Yaskawa INFORM job: A_ROOF_SIDE_0617_2_PAINT_60.JBI

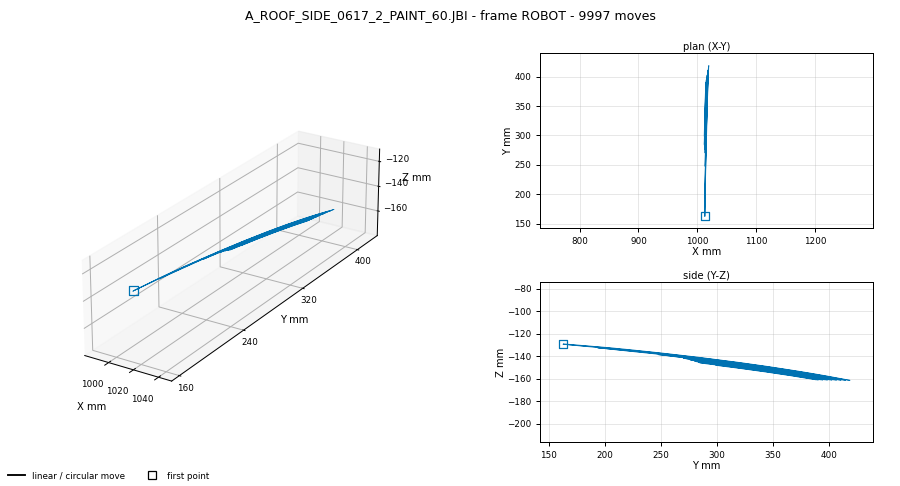
[picture p0: tool path of A_ROOF_SIDE_0617_2_PAINT_60.JBI in frame ROBOT, 9997 of 9997 moves have a stored position in this frame; points joined in program order, loops and branches not executed]
/JOB
//NAME A_ROOF_SIDE_0617_2_PAINT60
//POS
///NPOS 9997,0,0,0,0,0
///TOOL 1
///USER 0
///POSTYPE ROBOT
///RECTAN
///RCONF 1,0,0,0,0,0,0,0,0,0,0,0,0,0,0,0,0,0,0,0,0,0,0,0
C00000=1012.766,163.201,-128.936,166.543,56.945,160.429
C00001=1012.769,163.450,-128.956,166.546,56.934,160.427
C00002=1012.773,163.699,-128.974,166.549,56.922,160.426
C00003=1012.776,163.949,-128.994,166.553,56.910,160.424
C00004=1012.781,164.198,-129.014,166.556,56.898,160.423
C00005=1012.783,164.447,-129.033,166.560,56.886,160.421
C00006=1012.788,164.696,-129.052,166.563,56.875,160.420
C00007=1012.791,164.945,-129.072,166.568,56.863,160.418
C00008=1012.795,165.195,-129.092,166.571,56.851,160.417
C00009=1012.798,165.444,-129.111,166.574,56.839,160.415
C00010=1012.802,165.693,-129.131,166.578,56.827,160.414
C00011=1012.806,165.942,-129.150,166.581,56.815,160.412
C00012=1012.810,166.191,-129.170,166.586,56.803,160.411
C00013=1012.813,166.441,-129.189,166.589,56.791,160.409
C00014=1012.817,166.690,-129.209,166.592,56.779,160.408
C00015=1012.820,166.939,-129.229,166.596,56.767,160.406
C00016=1012.825,167.188,-129.248,166.599,56.756,160.405
C00017=1012.828,167.437,-129.267,166.604,56.743,160.403
C00018=1012.832,167.686,-129.287,166.607,56.732,160.402
C00019=1012.836,167.936,-129.307,166.610,56.720,160.400
C00020=1012.839,168.185,-129.327,166.614,56.707,160.398
C00021=1012.843,168.434,-129.346,166.617,56.695,160.397
C00022=1012.846,168.684,-129.365,166.621,56.683,160.395
C00023=1012.851,168.933,-129.385,166.624,56.671,160.394
C00024=1012.854,169.182,-129.405,166.629,56.659,160.393
C00025=1012.858,169.431,-129.425,166.632,56.647,160.391
C00026=1012.862,169.680,-129.444,166.636,56.635,160.390
C00027=1012.866,169.930,-129.464,166.639,56.623,160.388
C00028=1012.870,170.208,-129.486,166.644,56.609,160.386
C00029=1012.874,170.487,-129.508,166.648,56.596,160.385
C00030=1012.878,170.766,-129.530,166.652,56.583,160.383
C00031=1012.882,171.045,-129.552,166.656,56.569,160.381
C00032=1012.887,171.294,-129.572,166.661,56.557,160.380
C00033=1012.890,171.543,-129.592,166.664,56.545,160.378
C00034=1012.894,171.793,-129.611,166.668,56.532,160.377
C00035=1012.898,172.042,-129.631,166.671,56.521,160.375
C00036=1012.902,172.292,-129.651,166.675,56.509,160.374
C00037=1012.906,172.541,-129.670,166.678,56.497,160.372
C00038=1012.910,172.790,-129.690,166.683,56.485,160.371
C00039=1012.913,173.040,-129.710,166.687,56.472,160.369
C00040=1012.917,173.288,-129.729,166.690,56.460,160.367
C00041=1012.921,173.537,-129.749,166.694,56.448,160.366
C00042=1012.925,173.786,-129.769,166.699,56.436,160.365
C00043=1012.928,174.036,-129.789,166.701,56.424,160.363
C00044=1012.932,174.285,-129.809,166.706,56.411,160.361
C00045=1012.936,174.534,-129.828,166.710,56.399,160.360
C00046=1012.940,174.783,-129.849,166.713,56.388,160.358
C00047=1012.944,175.032,-129.868,166.717,56.375,160.357
C00048=1012.948,175.282,-129.888,166.721,56.363,160.355
C00049=1012.952,175.531,-129.908,166.725,56.351,160.354
C00050=1012.956,175.780,-129.928,166.729,56.339,160.352
C00051=1012.960,176.030,-129.948,166.733,56.326,160.351
C00052=1012.964,176.279,-129.967,166.737,56.314,160.349
C00053=1012.968,176.527,-129.988,166.741,56.302,160.348
C00054=1012.972,176.776,-130.007,166.744,56.289,160.346
C00055=1012.976,177.026,-130.027,166.749,56.277,160.345
C00056=1012.979,177.275,-130.048,166.753,56.265,160.343
C00057=1012.984,177.524,-130.067,166.757,56.252,160.342
C00058=1012.987,177.773,-130.087,166.760,56.241,160.340
C00059=1012.992,178.022,-130.107,166.765,56.229,160.339
C00060=1012.995,178.272,-130.127,166.769,56.216,160.337
C00061=1012.999,178.521,-130.147,166.773,56.204,160.336
C00062=1013.004,178.770,-130.167,166.777,56.191,160.334
C00063=1013.007,179.019,-130.187,166.780,56.179,160.332
C00064=1013.012,179.268,-130.206,166.785,56.167,160.331
C00065=1013.015,179.517,-130.226,166.788,56.155,160.329
C00066=1013.019,179.767,-130.247,166.793,56.142,160.328
C00067=1013.023,180.016,-130.266,166.797,56.130,160.326
C00068=1013.028,180.265,-130.287,166.801,56.118,160.325
C00069=1013.032,180.514,-130.307,166.805,56.105,160.323
C00070=1013.036,180.764,-130.327,166.809,56.093,160.322
C00071=1013.039,181.013,-130.347,166.813,56.081,160.320
C00072=1013.044,181.261,-130.367,166.817,56.068,160.319
C00073=1013.047,181.511,-130.387,166.821,56.056,160.317
C00074=1013.050,181.760,-130.408,166.826,56.044,160.316
C00075=1013.055,182.010,-130.429,166.830,56.032,160.314
C00076=1013.059,182.259,-130.450,166.833,56.020,160.313
C00077=1013.062,182.508,-130.470,166.837,56.008,160.311
C00078=1013.066,182.757,-130.491,166.842,55.996,160.310
C00079=1013.069,183.006,-130.511,166.846,55.984,160.309
C00080=1013.073,183.255,-130.532,166.849,55.972,160.307
C00081=1013.076,183.504,-130.553,166.854,55.960,160.306
C00082=1013.080,183.753,-130.573,166.858,55.947,160.304
C00083=1013.084,184.003,-130.594,166.863,55.935,160.303
C00084=1013.088,184.252,-130.615,166.866,55.924,160.301
C00085=1013.091,184.501,-130.637,166.870,55.911,160.300
C00086=1013.095,184.750,-130.657,166.874,55.899,160.298
C00087=1013.099,184.999,-130.677,166.879,55.887,160.297
C00088=1013.103,185.247,-130.698,166.883,55.874,160.295
C00089=1013.106,185.497,-130.719,166.887,55.862,160.294
C00090=1013.110,185.747,-130.740,166.891,55.851,160.292
C00091=1013.114,185.995,-130.761,166.895,55.839,160.291
C00092=1013.118,186.274,-130.784,166.900,55.825,160.289
C00093=1013.122,186.553,-130.808,166.904,55.811,160.287
C00094=1013.127,186.832,-130.831,166.910,55.798,160.286
C00095=1013.131,187.111,-130.854,166.915,55.784,160.284
C00096=1013.134,187.360,-130.875,166.918,55.772,160.283
C00097=1013.139,187.610,-130.896,166.922,55.759,160.281
C00098=1013.142,187.858,-130.917,166.927,55.748,160.280
C00099=1013.146,188.107,-130.937,166.931,55.736,160.278
C00100=1013.150,188.356,-130.959,166.935,55.723,160.277
C00101=1013.154,188.606,-130.980,166.940,55.711,160.275
C00102=1013.158,188.854,-131.001,166.944,55.699,160.274
C00103=1013.162,189.103,-131.021,166.948,55.686,160.272
C00104=1013.165,189.353,-131.042,166.953,55.674,160.271
C00105=1013.169,189.602,-131.063,166.957,55.662,160.270
C00106=1013.173,189.851,-131.084,166.961,55.650,160.268
C00107=1013.176,190.100,-131.105,166.966,55.638,160.267
C00108=1013.181,190.349,-131.126,166.970,55.625,160.265
C00109=1013.185,190.598,-131.147,166.975,55.613,160.264
C00110=1013.189,190.847,-131.168,166.979,55.601,160.262
C00111=1013.192,191.097,-131.190,166.983,55.588,160.261
C00112=1013.196,191.345,-131.211,166.988,55.576,160.259
C00113=1013.200,191.594,-131.231,166.992,55.564,160.258
C00114=1013.205,191.843,-131.253,166.996,55.552,160.256
C00115=1013.208,192.092,-131.274,167.001,55.540,160.255
C00116=1013.212,192.341,-131.295,167.005,55.527,160.253
C00117=1013.216,192.591,-131.316,167.010,55.515,160.252
C00118=1013.220,192.840,-131.337,167.015,55.502,160.251
C00119=1013.224,193.088,-131.358,167.019,55.490,160.249
C00120=1013.228,193.338,-131.379,167.023,55.478,160.248
C00121=1013.232,193.587,-131.400,167.028,55.466,160.246
C00122=1013.236,193.836,-131.422,167.033,55.454,160.245
C00123=1013.240,194.085,-131.442,167.037,55.441,160.243
C00124=1013.244,194.334,-131.463,167.041,55.429,160.242
C00125=1013.248,194.583,-131.484,167.045,55.417,160.240
C00126=1013.251,194.832,-131.506,167.051,55.404,160.239
C00127=1013.256,195.082,-131.527,167.055,55.392,160.237
C00128=1013.260,195.330,-131.548,167.060,55.380,160.236
C00129=1013.263,195.580,-131.569,167.064,55.367,160.234
C00130=1013.267,195.829,-131.590,167.068,55.355,160.233
C00131=1013.271,196.078,-131.611,167.073,55.343,160.231
C00132=1013.276,196.326,-131.633,167.078,55.331,160.230
C00133=1013.279,196.576,-131.654,167.082,55.318,160.229
C00134=1013.284,196.825,-131.675,167.087,55.306,160.227
C00135=1013.288,197.074,-131.696,167.091,55.293,160.226
C00136=1013.292,197.323,-131.717,167.097,55.281,160.224
C00137=1013.295,197.572,-131.739,167.101,55.269,160.223
C00138=1013.300,197.821,-131.761,167.106,55.257,160.221
C00139=1013.304,198.070,-131.781,167.110,55.244,160.220
C00140=1013.308,198.319,-131.803,167.115,55.232,160.219
C00141=1013.312,198.568,-131.824,167.120,55.219,160.217
C00142=1013.316,198.818,-131.845,167.124,55.207,160.216
C00143=1013.320,199.067,-131.867,167.128,55.195,160.214
C00144=1013.324,199.316,-131.889,167.134,55.183,160.213
C00145=1013.328,199.565,-131.911,167.138,55.170,160.211
C00146=1013.332,199.814,-131.932,167.143,55.158,160.210
C00147=1013.336,200.063,-131.955,167.148,55.146,160.209
C00148=1013.340,200.312,-131.975,167.152,55.134,160.207
C00149=1013.344,200.561,-131.998,167.157,55.122,160.206
C00150=1013.347,200.810,-132.019,167.162,55.109,160.204
C00151=1013.352,201.059,-132.041,167.166,55.097,160.203
C00152=1013.356,201.308,-132.063,167.171,55.085,160.201
C00153=1013.359,201.557,-132.085,167.176,55.072,160.200
C00154=1013.364,201.806,-132.106,167.181,55.061,160.199
C00155=1013.367,202.055,-132.128,167.185,55.048,160.197
C00156=1013.384,203.102,-132.220,167.720,55.151,160.345
C00157=1013.390,203.386,-132.246,167.725,55.138,160.343
C00158=1013.395,203.671,-132.273,167.730,55.125,160.342
C00159=1013.402,203.957,-132.300,167.736,55.113,160.340
C00160=1013.408,204.241,-132.328,167.741,55.100,160.339
C00161=1013.412,204.490,-132.351,167.746,55.089,160.337
C00162=1013.417,204.739,-132.374,167.751,55.077,160.336
C00163=1013.422,204.988,-132.398,167.755,55.066,160.335
C00164=1013.428,205.237,-132.421,167.760,55.055,160.333
C00165=1013.433,205.486,-132.445,167.764,55.045,160.332
C00166=1013.438,205.734,-132.469,167.769,55.034,160.331
C00167=1013.443,205.983,-132.492,167.773,55.022,160.329
C00168=1013.448,206.232,-132.516,167.778,55.011,160.328
C00169=1013.453,206.481,-132.540,167.782,55.001,160.327
C00170=1013.458,206.730,-132.564,167.787,54.989,160.326
C00171=1013.463,206.978,-132.588,167.791,54.979,160.324
C00172=1013.468,207.227,-132.611,167.796,54.968,160.323
C00173=1013.473,207.476,-132.635,167.800,54.957,160.322
C00174=1013.478,207.725,-132.659,167.806,54.946,160.320
C00175=1013.483,207.973,-132.683,167.810,54.935,160.319
C00176=1013.488,208.223,-132.707,167.815,54.924,160.318
C00177=1013.493,208.451,-132.729,167.818,54.914,160.316
C00178=1013.498,208.678,-132.750,167.822,54.904,160.315
C00179=1013.502,208.907,-132.772,167.827,54.894,160.314
C00180=1013.507,209.134,-132.794,167.831,54.885,160.313
C00181=1013.511,209.362,-132.816,167.835,54.875,160.312
C00182=1013.516,209.590,-132.839,167.840,54.865,160.311
C00183=1013.520,209.818,-132.861,167.844,54.855,160.310
C00184=1013.525,210.046,-132.882,167.848,54.845,160.309
C00185=1013.530,210.294,-132.907,167.852,54.835,160.307
C00186=1013.535,210.544,-132.931,167.856,54.824,160.306
C00187=1013.540,210.792,-132.955,167.862,54.813,160.305
C00188=1013.545,211.041,-132.979,167.866,54.802,160.303
C00189=1013.550,211.290,-133.003,167.871,54.791,160.302
C00190=1013.555,211.539,-133.028,167.875,54.781,160.301
C00191=1013.560,211.788,-133.052,167.880,54.771,160.300
C00192=1013.565,212.036,-133.076,167.885,54.760,160.299
C00193=1013.570,212.285,-133.100,167.889,54.749,160.297
C00194=1013.576,212.534,-133.124,167.893,54.739,160.296
C00195=1013.580,212.783,-133.149,167.898,54.728,160.295
C00196=1013.586,213.032,-133.173,167.903,54.718,160.294
C00197=1013.591,213.280,-133.197,167.907,54.707,160.292
C00198=1013.596,213.529,-133.221,167.911,54.697,160.291
C00199=1013.601,213.778,-133.245,167.917,54.686,160.290
C00200=1013.606,214.027,-133.270,167.921,54.676,160.289
C00201=1013.611,214.275,-133.294,167.925,54.665,160.287
C00202=1013.616,214.524,-133.319,167.931,54.654,160.286
C00203=1013.622,214.773,-133.343,167.935,54.644,160.285
C00204=1013.626,215.021,-133.368,167.939,54.634,160.284
C00205=1013.631,215.271,-133.391,167.944,54.623,160.282
C00206=1013.636,215.519,-133.415,167.949,54.613,160.281
C00207=1013.642,215.769,-133.440,167.954,54.602,160.280
C00208=1013.648,216.017,-133.464,167.958,54.592,160.279
C00209=1013.652,216.266,-133.489,167.963,54.581,160.278
C00210=1013.657,216.515,-133.513,167.968,54.571,160.277
C00211=1013.663,216.763,-133.538,167.972,54.561,160.275
C00212=1013.668,217.012,-133.562,167.977,54.550,160.274
C00213=1013.673,217.261,-133.587,167.982,54.539,160.273
C00214=1013.678,217.509,-133.611,167.987,54.529,160.272
C00215=1013.683,217.758,-133.635,167.991,54.519,160.271
C00216=1013.688,218.007,-133.660,167.995,54.509,160.269
C00217=1013.694,218.258,-133.685,168.000,54.498,160.268
C00218=1013.699,218.511,-133.711,168.005,54.488,160.267
C00219=1013.704,218.764,-133.736,168.010,54.478,160.266
C00220=1013.709,219.015,-133.761,168.014,54.468,160.265
C00221=1013.714,219.263,-133.785,168.019,54.457,160.263
C00222=1013.719,219.513,-133.811,168.023,54.447,160.262
C00223=1013.724,219.762,-133.835,168.028,54.437,160.261
C00224=1013.729,220.010,-133.860,168.033,54.427,160.260
C00225=1013.735,220.259,-133.885,168.038,54.417,160.259
C00226=1013.739,220.507,-133.910,168.043,54.407,160.258
C00227=1013.745,220.757,-133.934,168.047,54.396,160.257
C00228=1013.750,221.005,-133.960,168.052,54.386,160.256
C00229=1013.755,221.254,-133.984,168.056,54.377,160.254
C00230=1013.760,221.503,-134.009,168.061,54.367,160.253
C00231=1013.765,221.750,-134.034,168.065,54.356,160.252
C00232=1013.770,222.000,-134.059,168.070,54.346,160.251
C00233=1013.776,222.249,-134.083,168.075,54.337,160.250
C00234=1013.781,222.497,-134.109,168.080,54.327,160.249
C00235=1013.786,222.746,-134.133,168.084,54.316,160.247
C00236=1013.791,222.995,-134.158,168.090,54.306,160.247
C00237=1013.797,223.243,-134.183,168.094,54.296,160.245
C00238=1013.801,223.492,-134.208,168.099,54.286,160.244
C00239=1013.807,223.741,-134.233,168.104,54.277,160.243
C00240=1013.812,223.990,-134.258,168.108,54.266,160.242
C00241=1013.817,224.238,-134.283,168.113,54.256,160.241
C00242=1013.823,224.487,-134.308,168.118,54.246,160.240
C00243=1013.827,224.736,-134.333,168.122,54.237,160.239
C00244=1013.833,224.984,-134.358,168.127,54.227,160.238
C00245=1013.838,225.234,-134.384,168.132,54.217,160.237
C00246=1013.844,225.482,-134.408,168.137,54.207,160.236
C00247=1013.848,225.730,-134.433,168.141,54.197,160.234
C00248=1013.854,225.979,-134.459,168.146,54.187,160.233
C00249=1013.859,226.228,-134.484,168.151,54.177,160.232
C00250=1013.864,226.476,-134.509,168.156,54.168,160.231
C00251=1013.869,226.725,-134.535,168.161,54.158,160.230
C00252=1013.875,226.974,-134.559,168.165,54.148,160.229
C00253=1013.880,227.223,-134.585,168.170,54.139,160.228
C00254=1013.885,227.471,-134.611,168.174,54.129,160.227
C00255=1013.890,227.720,-134.636,168.179,54.119,160.226
C00256=1013.895,227.969,-134.662,168.184,54.110,160.225
C00257=1013.901,228.217,-134.687,168.188,54.100,160.224
C00258=1013.906,228.466,-134.712,168.193,54.090,160.222
C00259=1013.911,228.715,-134.737,168.198,54.080,160.221
C00260=1013.916,228.963,-134.763,168.203,54.071,160.221
C00261=1013.922,229.212,-134.788,168.208,54.061,160.219
C00262=1013.927,229.460,-134.814,168.213,54.052,160.218
C00263=1013.932,229.709,-134.840,168.217,54.042,160.217
C00264=1013.937,229.957,-134.865,168.222,54.033,160.216
C00265=1013.942,230.206,-134.890,168.227,54.023,160.215
C00266=1013.947,230.455,-134.916,168.231,54.014,160.214
C00267=1013.952,230.704,-134.942,168.236,54.004,160.213
C00268=1013.957,230.952,-134.968,168.242,53.995,160.212
C00269=1013.962,231.201,-134.993,168.245,53.985,160.211
C00270=1013.968,231.450,-135.019,168.250,53.976,160.210
C00271=1013.973,231.698,-135.045,168.256,53.967,160.209
C00272=1013.978,231.947,-135.071,168.260,53.957,160.208
C00273=1013.983,232.195,-135.096,168.265,53.947,160.207
C00274=1013.989,232.444,-135.121,168.269,53.938,160.206
C00275=1013.994,232.692,-135.147,168.274,53.929,160.205
C00276=1013.999,232.941,-135.173,168.280,53.920,160.204
C00277=1014.005,233.188,-135.198,168.284,53.910,160.203
C00278=1014.010,233.433,-135.224,168.289,53.901,160.202
C00279=1014.014,233.680,-135.250,168.294,53.892,160.201
C00280=1014.020,233.927,-135.275,168.299,53.882,160.200
C00281=1014.025,234.173,-135.301,168.303,53.873,160.199
C00282=1014.030,234.419,-135.326,168.308,53.864,160.198
C00283=1014.036,234.665,-135.352,168.313,53.854,160.197
C00284=1014.041,234.911,-135.378,168.317,53.846,160.196
C00285=1014.046,235.159,-135.403,168.322,53.836,160.195
C00286=1014.051,235.408,-135.429,168.327,53.827,160.194
C00287=1014.057,235.657,-135.456,168.333,53.818,160.193
C00288=1014.062,235.905,-135.481,168.336,53.809,160.192
C00289=1014.067,236.154,-135.507,168.342,53.800,160.191
C00290=1014.073,236.403,-135.533,168.347,53.790,160.190
C00291=1014.078,236.651,-135.559,168.351,53.781,160.189
C00292=1014.083,236.900,-135.585,168.356,53.772,160.189
C00293=1014.089,237.149,-135.611,168.361,53.762,160.187
C00294=1014.094,237.397,-135.637,168.365,53.754,160.186
C00295=1014.099,237.646,-135.663,168.370,53.744,160.185
C00296=1014.105,237.894,-135.689,168.376,53.735,160.185
C00297=1014.110,238.143,-135.715,168.381,53.726,160.184
C00298=1014.115,238.392,-135.741,168.385,53.717,160.183
C00299=1014.121,238.639,-135.767,168.390,53.708,160.182
C00300=1014.126,238.888,-135.793,168.395,53.699,160.181
C00301=1014.131,239.137,-135.820,168.400,53.690,160.180
C00302=1014.136,239.386,-135.846,168.405,53.681,160.179
C00303=1014.142,239.633,-135.873,168.410,53.673,160.178
C00304=1014.146,239.883,-135.899,168.414,53.663,160.177
C00305=1014.152,240.131,-135.926,168.419,53.654,160.176
C00306=1014.157,240.379,-135.951,168.424,53.645,160.175
C00307=1014.163,240.628,-135.978,168.430,53.636,160.174
C00308=1014.168,240.877,-136.005,168.434,53.628,160.173
C00309=1014.173,241.125,-136.031,168.439,53.619,160.173
C00310=1014.178,241.374,-136.057,168.444,53.610,160.172
C00311=1014.183,241.622,-136.084,168.449,53.601,160.171
C00312=1014.189,241.871,-136.111,168.453,53.592,160.170
C00313=1014.194,242.120,-136.137,168.459,53.583,160.169
C00314=1014.200,242.367,-136.163,168.464,53.574,160.168
C00315=1014.205,242.616,-136.190,168.468,53.566,160.167
C00316=1014.210,242.865,-136.216,168.474,53.557,160.166
C00317=1014.215,243.114,-136.243,168.478,53.548,160.165
C00318=1014.221,243.362,-136.270,168.482,53.540,160.164
C00319=1014.225,243.610,-136.297,168.488,53.531,160.164
C00320=1014.231,243.858,-136.323,168.493,53.523,160.163
C00321=1014.236,244.107,-136.351,168.498,53.514,160.162
C00322=1014.241,244.356,-136.377,168.502,53.505,160.161
C00323=1014.247,244.605,-136.404,168.508,53.496,160.160
C00324=1014.252,244.853,-136.431,168.512,53.488,160.159
C00325=1014.257,245.101,-136.457,168.518,53.479,160.159
C00326=1014.262,245.350,-136.485,168.522,53.471,160.158
C00327=1014.267,245.598,-136.512,168.527,53.462,160.157
C00328=1014.273,245.847,-136.539,168.532,53.453,160.156
C00329=1014.278,246.095,-136.566,168.537,53.445,160.155
C00330=1014.284,246.344,-136.592,168.542,53.436,160.154
C00331=1014.289,246.592,-136.620,168.547,53.428,160.153
C00332=1014.294,246.841,-136.647,168.553,53.420,160.153
C00333=1014.299,247.089,-136.674,168.557,53.411,160.152
C00334=1014.304,247.337,-136.700,168.561,53.403,160.151
C00335=1014.310,247.586,-136.727,168.567,53.394,160.150
C00336=1014.315,247.834,-136.754,168.572,53.386,160.149
C00337=1014.320,248.077,-136.780,168.577,53.378,160.149
C00338=1014.325,248.321,-136.807,168.582,53.369,160.148
C00339=1014.331,248.563,-136.833,168.587,53.361,160.147
C00340=1014.336,248.806,-136.860,168.591,53.352,160.146
C00341=1014.341,249.049,-136.885,168.596,53.345,160.145
C00342=1014.346,249.291,-136.913,168.600,53.336,160.144
C00343=1014.352,249.534,-136.939,168.606,53.328,160.144
C00344=1014.356,249.777,-136.965,168.611,53.320,160.143
C00345=1014.362,250.025,-136.992,168.616,53.311,160.142
C00346=1014.367,250.274,-137.019,168.621,53.303,160.142
C00347=1014.373,250.522,-137.047,168.626,53.295,160.141
C00348=1014.378,250.770,-137.074,168.631,53.287,160.140
C00349=1014.383,251.019,-137.101,168.636,53.278,160.139
C00350=1014.389,251.267,-137.128,168.641,53.270,160.138
C00351=1014.394,251.516,-137.155,168.645,53.261,160.137
C00352=1014.400,251.765,-137.183,168.651,53.253,160.137
C00353=1014.406,252.013,-137.210,168.656,53.245,160.136
C00354=1014.411,252.262,-137.237,168.662,53.236,160.135
C00355=1014.417,252.510,-137.264,168.667,53.229,160.134
C00356=1014.422,252.759,-137.291,168.671,53.220,160.134
C00357=1014.427,253.007,-137.319,168.677,53.212,160.133
C00358=1014.433,253.255,-137.346,168.681,53.203,160.132
C00359=1014.438,253.504,-137.373,168.686,53.195,160.131
C00360=1014.444,253.752,-137.400,168.692,53.187,160.131
C00361=1014.450,254.001,-137.428,168.696,53.179,160.130
C00362=1014.455,254.250,-137.455,168.701,53.171,160.129
C00363=1014.461,254.497,-137.483,168.707,53.163,160.128
C00364=1014.466,254.746,-137.510,168.712,53.155,160.128
C00365=1014.472,254.994,-137.536,168.717,53.146,160.127
C00366=1014.477,255.243,-137.564,168.722,53.138,160.126
C00367=1014.483,255.492,-137.592,168.727,53.130,160.125
C00368=1014.489,255.740,-137.619,168.732,53.122,160.124
C00369=1014.494,255.988,-137.647,168.738,53.114,160.124
C00370=1014.499,256.237,-137.673,168.743,53.106,160.123
C00371=1014.505,256.485,-137.702,168.747,53.098,160.122
C00372=1014.510,256.734,-137.729,168.753,53.090,160.122
C00373=1014.516,256.982,-137.756,168.758,53.081,160.121
C00374=1014.522,257.231,-137.783,168.763,53.073,160.120
C00375=1014.527,257.479,-137.812,168.768,53.066,160.119
C00376=1014.533,257.728,-137.838,168.773,53.057,160.119
C00377=1014.539,257.976,-137.866,168.778,53.050,160.118
C00378=1014.545,258.225,-137.893,168.783,53.042,160.117
C00379=1014.550,258.473,-137.921,168.789,53.034,160.117
C00380=1014.555,258.721,-137.949,168.794,53.026,160.116
C00381=1014.561,258.969,-137.976,168.799,53.017,160.115
C00382=1014.567,259.218,-138.004,168.803,53.009,160.114
C00383=1014.573,259.466,-138.032,168.809,53.001,160.114
C00384=1014.578,259.714,-138.059,168.814,52.993,160.113
C00385=1014.584,259.962,-138.087,168.820,52.986,160.112
C00386=1014.590,260.211,-138.115,168.825,52.979,160.112
C00387=1014.595,260.459,-138.143,168.829,52.971,160.111
C00388=1014.600,260.707,-138.171,168.835,52.963,160.110
C00389=1014.606,260.956,-138.199,168.840,52.955,160.110
C00390=1014.611,261.205,-138.227,168.845,52.947,160.109
C00391=1014.617,261.453,-138.255,168.851,52.940,160.108
C00392=1014.623,261.701,-138.283,168.856,52.932,160.108
C00393=1014.627,261.950,-138.311,168.860,52.924,160.107
C00394=1014.633,262.198,-138.339,168.865,52.916,160.106
C00395=1014.639,262.447,-138.368,168.872,52.909,160.106
C00396=1014.644,262.695,-138.396,168.877,52.901,160.105
C00397=1014.650,262.936,-138.423,168.882,52.893,160.104
C00398=1014.655,263.178,-138.450,168.887,52.886,160.104
C00399=1014.660,263.420,-138.478,168.892,52.879,160.103
C00400=1014.666,263.662,-138.505,168.896,52.872,160.102
C00401=1014.671,263.903,-138.533,168.901,52.864,160.102
C00402=1014.677,264.146,-138.560,168.907,52.857,160.101
C00403=1014.682,264.387,-138.587,168.912,52.849,160.100
C00404=1014.687,264.629,-138.615,168.917,52.842,160.100
C00405=1014.693,264.877,-138.644,168.922,52.834,160.099
C00406=1014.699,265.125,-138.672,168.927,52.827,160.099
C00407=1014.705,265.374,-138.700,168.932,52.819,160.098
C00408=1014.710,265.622,-138.728,168.938,52.812,160.097
C00409=1014.716,265.871,-138.757,168.944,52.804,160.097
C00410=1014.721,266.119,-138.785,168.949,52.797,160.096
C00411=1014.727,266.367,-138.814,168.954,52.789,160.096
C00412=1014.732,266.615,-138.842,168.959,52.782,160.095
C00413=1014.738,266.864,-138.871,168.964,52.774,160.094
C00414=1014.744,267.112,-138.899,168.970,52.767,160.094
C00415=1014.749,267.361,-138.928,168.975,52.760,160.093
C00416=1014.755,267.608,-138.956,168.980,52.753,160.093
C00417=1014.761,267.857,-138.985,168.985,52.745,160.092
C00418=1014.767,268.106,-139.013,168.990,52.738,160.091
C00419=1014.771,268.353,-139.042,168.996,52.731,160.091
C00420=1014.777,268.602,-139.071,169.001,52.724,160.090
C00421=1014.783,268.850,-139.099,169.006,52.716,160.090
C00422=1014.789,269.098,-139.128,169.011,52.709,160.089
C00423=1014.794,269.347,-139.156,169.017,52.702,160.089
C00424=1014.800,269.595,-139.185,169.022,52.695,160.088
C00425=1014.806,269.844,-139.213,169.027,52.687,160.087
C00426=1014.811,270.091,-139.243,169.033,52.680,160.087
C00427=1014.817,270.340,-139.271,169.038,52.673,160.086
C00428=1014.822,270.588,-139.301,169.043,52.666,160.086
C00429=1014.827,270.837,-139.329,169.049,52.659,160.085
C00430=1014.834,271.085,-139.358,169.054,52.652,160.085
C00431=1014.839,271.332,-139.387,169.059,52.644,160.084
C00432=1014.845,271.581,-139.415,169.065,52.637,160.084
C00433=1014.851,271.829,-139.444,169.070,52.630,160.083
C00434=1014.856,272.077,-139.474,169.075,52.623,160.083
C00435=1014.862,272.326,-139.502,169.081,52.616,160.082
C00436=1014.867,272.574,-139.532,169.086,52.608,160.082
C00437=1014.873,272.822,-139.561,169.092,52.601,160.081
C00438=1014.878,273.071,-139.589,169.097,52.594,160.081
C00439=1014.884,273.319,-139.618,169.102,52.587,160.080
C00440=1014.890,273.567,-139.648,169.108,52.580,160.080
C00441=1014.895,273.815,-139.677,169.113,52.573,160.079
C00442=1014.901,274.064,-139.705,169.119,52.566,160.079
C00443=1014.907,274.312,-139.734,169.124,52.559,160.078
C00444=1014.913,274.560,-139.764,169.129,52.552,160.078
C00445=1014.918,274.808,-139.793,169.135,52.545,160.077
C00446=1014.924,275.056,-139.822,169.140,52.538,160.077
C00447=1014.930,275.304,-139.851,169.146,52.531,160.076
C00448=1014.936,275.553,-139.880,169.151,52.524,160.076
C00449=1014.941,275.802,-139.909,169.157,52.517,160.075
C00450=1014.947,276.049,-139.938,169.162,52.511,160.075
C00451=1014.952,276.297,-139.968,169.168,52.504,160.074
C00452=1014.958,276.546,-139.997,169.172,52.497,160.074
C00453=1014.964,276.794,-140.026,169.178,52.490,160.073
C00454=1014.970,277.042,-140.057,169.184,52.483,160.073
C00455=1014.975,277.290,-140.086,169.189,52.476,160.072
C00456=1014.980,277.538,-140.116,169.194,52.469,160.072
C00457=1014.986,277.782,-140.144,169.200,52.463,160.072
C00458=1014.992,278.027,-140.173,169.205,52.456,160.071
C00459=1014.998,278.270,-140.202,169.211,52.450,160.071
C00460=1015.003,278.514,-140.231,169.216,52.443,160.070
C00461=1015.009,278.758,-140.261,169.222,52.437,160.070
C00462=1015.014,279.002,-140.290,169.226,52.430,160.069
C00463=1015.020,279.247,-140.318,169.232,52.424,160.069
C00464=1015.026,279.490,-140.348,169.238,52.417,160.068
C00465=1015.031,279.739,-140.378,169.243,52.410,160.068
C00466=1015.038,279.987,-140.407,169.249,52.403,160.068
C00467=1015.043,280.235,-140.437,169.254,52.396,160.067
C00468=1015.049,280.483,-140.467,169.259,52.390,160.067
C00469=1015.054,280.732,-140.496,169.265,52.383,160.066
C00470=1015.061,280.980,-140.525,169.270,52.377,160.066
C00471=1015.067,281.228,-140.556,169.276,52.370,160.065
C00472=1015.072,281.476,-140.585,169.282,52.364,160.065
C00473=1015.077,281.724,-140.614,169.287,52.357,160.065
C00474=1015.084,281.972,-140.645,169.293,52.350,160.064
C00475=1015.090,282.220,-140.674,169.298,52.344,160.064
C00476=1015.095,282.469,-140.704,169.303,52.337,160.063
C00477=1015.102,282.716,-140.734,169.309,52.331,160.063
C00478=1015.107,282.965,-140.763,169.315,52.324,160.063
C00479=1015.113,283.213,-140.794,169.321,52.318,160.062
C00480=1015.119,283.461,-140.823,169.326,52.311,160.062
C00481=1015.125,283.709,-140.853,169.332,52.304,160.061
C00482=1015.131,283.957,-140.883,169.337,52.298,160.061
C00483=1015.136,284.205,-140.913,169.343,52.292,160.061
C00484=1015.142,284.453,-140.943,169.348,52.285,160.060
C00485=1015.148,284.701,-140.973,169.354,52.279,160.060
C00486=1015.154,284.949,-141.003,169.360,52.272,160.060
C00487=1015.159,285.197,-141.033,169.366,52.266,160.059
C00488=1015.166,285.445,-141.063,169.370,52.259,160.059
C00489=1015.171,285.693,-141.093,169.376,52.253,160.058
C00490=1015.178,285.942,-141.123,169.382,52.247,160.058
C00491=1015.183,286.190,-141.153,169.388,52.240,160.058
C00492=1015.189,286.438,-141.184,169.394,52.234,160.058
C00493=1015.195,286.686,-141.213,169.399,52.228,160.057
C00494=1015.201,286.934,-141.244,169.405,52.222,160.057
C00495=1015.206,287.182,-141.274,169.410,52.216,160.057
C00496=1015.212,287.429,-141.304,169.416,52.209,160.056
C00497=1015.219,287.678,-141.335,169.422,52.203,160.056
C00498=1015.224,287.926,-141.366,169.427,52.197,160.056
C00499=1015.230,288.174,-141.395,169.433,52.191,160.055
C00500=1015.236,288.422,-141.425,169.439,52.184,160.055
C00501=1015.242,288.670,-141.456,169.445,52.178,160.055
C00502=1015.248,288.918,-141.487,169.450,52.172,160.054
C00503=1015.254,289.166,-141.517,169.456,52.166,160.054
C00504=1015.259,289.414,-141.548,169.461,52.160,160.054
C00505=1015.265,289.662,-141.578,169.467,52.153,160.053
C00506=1015.271,289.911,-141.609,169.472,52.147,160.053
C00507=1015.277,290.159,-141.639,169.478,52.141,160.053
C00508=1015.283,290.406,-141.670,169.484,52.135,160.052
C00509=1015.289,290.655,-141.700,169.490,52.128,160.052
C00510=1015.295,290.903,-141.731,169.496,52.123,160.052
C00511=1015.301,291.151,-141.761,169.501,52.117,160.052
C00512=1015.307,291.398,-141.791,169.507,52.111,160.051
C00513=1015.313,291.647,-141.822,169.513,52.104,160.051
C00514=1015.318,291.894,-141.854,169.519,52.099,160.051
C00515=1015.324,292.142,-141.884,169.524,52.093,160.050
C00516=1015.331,292.391,-141.915,169.530,52.086,160.050
C00517=1015.336,292.643,-141.946,169.536,52.080,160.050
C00518=1015.342,292.895,-141.978,169.542,52.075,160.050
C00519=1015.348,293.148,-142.009,169.548,52.068,160.049
C00520=1015.355,293.400,-142.041,169.553,52.063,160.049
C00521=1015.360,293.648,-142.072,169.559,52.057,160.049
C00522=1015.366,293.896,-142.103,169.566,52.051,160.049
C00523=1015.371,294.144,-142.134,169.571,52.045,160.049
C00524=1015.378,294.392,-142.165,169.577,52.040,160.048
C00525=1015.383,294.640,-142.196,169.583,52.033,160.048
C00526=1015.389,294.888,-142.228,169.588,52.028,160.048
C00527=1015.394,295.136,-142.258,169.594,52.022,160.048
C00528=1015.401,295.384,-142.290,169.600,52.016,160.048
C00529=1015.407,295.631,-142.322,169.606,52.011,160.047
C00530=1015.412,295.879,-142.352,169.612,52.005,160.047
C00531=1015.418,296.127,-142.384,169.618,51.999,160.047
C00532=1015.424,296.375,-142.414,169.623,51.993,160.047
C00533=1015.430,296.623,-142.446,169.629,51.987,160.046
C00534=1015.436,296.870,-142.477,169.636,51.982,160.046
C00535=1015.442,297.119,-142.509,169.640,51.976,160.046
C00536=1015.448,297.366,-142.540,169.647,51.970,160.046
C00537=1015.454,297.615,-142.572,169.653,51.965,160.046
C00538=1015.459,297.863,-142.603,169.658,51.960,160.046
C00539=1015.466,298.111,-142.634,169.664,51.953,160.045
C00540=1015.471,298.358,-142.666,169.671,51.948,160.045
C00541=1015.478,298.606,-142.697,169.676,51.942,160.045
C00542=1015.484,298.855,-142.729,169.682,51.937,160.045
C00543=1015.490,299.102,-142.760,169.688,51.931,160.045
C00544=1015.496,299.350,-142.792,169.694,51.925,160.044
C00545=1015.502,299.598,-142.823,169.700,51.920,160.044
C00546=1015.508,299.846,-142.854,169.706,51.914,160.044
C00547=1015.514,300.094,-142.885,169.712,51.909,160.044
C00548=1015.520,300.342,-142.917,169.718,51.903,160.044
C00549=1015.526,300.590,-142.949,169.724,51.898,160.044
C00550=1015.532,300.837,-142.980,169.729,51.892,160.044
C00551=1015.539,301.085,-143.012,169.736,51.886,160.043
C00552=1015.544,301.333,-143.044,169.742,51.881,160.043
C00553=1015.550,301.581,-143.075,169.747,51.875,160.043
C00554=1015.557,301.829,-143.107,169.754,51.870,160.043
C00555=1015.563,302.077,-143.139,169.760,51.864,160.043
C00556=1015.569,302.325,-143.170,169.765,51.859,160.043
C00557=1015.575,302.572,-143.202,169.772,51.853,160.043
C00558=1015.581,302.820,-143.233,169.778,51.848,160.043
C00559=1015.587,303.069,-143.265,169.783,51.843,160.042
C00560=1015.594,303.316,-143.297,169.790,51.837,160.042
C00561=1015.600,303.564,-143.328,169.796,51.831,160.042
C00562=1015.606,303.812,-143.360,169.802,51.826,160.042
C00563=1015.612,304.060,-143.392,169.808,51.821,160.042
C00564=1015.619,304.308,-143.423,169.814,51.816,160.042
C00565=1015.624,304.555,-143.455,169.821,51.810,160.042
C00566=1015.630,304.804,-143.487,169.826,51.805,160.042
C00567=1015.637,305.051,-143.519,169.832,51.799,160.042
C00568=1015.643,305.299,-143.551,169.839,51.794,160.042
C00569=1015.650,305.547,-143.583,169.844,51.789,160.041
C00570=1015.656,305.795,-143.615,169.851,51.784,160.042
C00571=1015.663,306.043,-143.646,169.857,51.778,160.041
C00572=1015.668,306.290,-143.678,169.863,51.773,160.041
C00573=1015.675,306.538,-143.710,169.869,51.767,160.041
C00574=1015.681,306.786,-143.742,169.876,51.762,160.041
C00575=1015.688,307.033,-143.774,169.882,51.757,160.041
C00576=1015.694,307.282,-143.806,169.887,51.752,160.041
C00577=1015.701,307.552,-143.841,169.895,51.746,160.041
C00578=1015.708,307.823,-143.876,169.901,51.740,160.041
C00579=1015.715,308.092,-143.911,169.907,51.735,160.041
C00580=1015.722,308.363,-143.946,169.915,51.729,160.041
C00581=1015.729,308.610,-143.978,169.922,51.724,160.041
C00582=1015.735,308.858,-144.010,169.927,51.719,160.041
C00583=1015.741,309.106,-144.041,169.933,51.713,160.041
C00584=1015.748,309.354,-144.074,169.940,51.708,160.041
C00585=1015.754,309.601,-144.107,169.945,51.703,160.040
C00586=1015.760,309.849,-144.139,169.952,51.698,160.041
C00587=1015.766,310.097,-144.172,169.958,51.693,160.041
C00588=1015.772,310.345,-144.205,169.964,51.688,160.040
C00589=1015.778,310.593,-144.238,169.970,51.683,160.041
C00590=1015.784,310.840,-144.270,169.977,51.678,160.041
C00591=1015.791,311.088,-144.303,169.984,51.674,160.041
C00592=1015.797,311.335,-144.336,169.989,51.668,160.041
C00593=1015.803,311.583,-144.369,169.996,51.663,160.041
C00594=1015.809,311.831,-144.401,170.001,51.659,160.041
C00595=1015.815,312.079,-144.434,170.008,51.654,160.041
C00596=1015.821,312.327,-144.467,170.015,51.648,160.041
C00597=1015.827,312.574,-144.499,170.020,51.644,160.041
C00598=1015.834,312.822,-144.532,170.027,51.639,160.041
C00599=1015.839,313.070,-144.566,170.033,51.635,160.041
C00600=1015.846,313.317,-144.598,170.040,51.630,160.041
C00601=1015.852,313.566,-144.631,170.046,51.625,160.041
C00602=1015.859,313.813,-144.665,170.052,51.620,160.041
C00603=1015.865,314.060,-144.698,170.059,51.615,160.041
C00604=1015.871,314.308,-144.731,170.065,51.611,160.041
C00605=1015.877,314.556,-144.764,170.072,51.606,160.041
C00606=1015.884,314.803,-144.796,170.078,51.600,160.041
C00607=1015.890,315.052,-144.830,170.084,51.596,160.041
C00608=1015.897,315.299,-144.862,170.090,51.591,160.041
C00609=1015.902,315.547,-144.896,170.096,51.586,160.041
C00610=1015.909,315.794,-144.929,170.103,51.582,160.042
C00611=1015.915,316.042,-144.962,170.110,51.577,160.042
C00612=1015.922,316.290,-144.995,170.116,51.573,160.042
C00613=1015.928,316.537,-145.028,170.123,51.568,160.042
C00614=1015.934,316.785,-145.062,170.129,51.563,160.042
C00615=1015.940,317.032,-145.094,170.135,51.558,160.042
C00616=1015.947,317.281,-145.128,170.142,51.554,160.042
C00617=1015.954,317.528,-145.161,170.148,51.549,160.042
C00618=1015.960,317.775,-145.194,170.155,51.544,160.042
C00619=1015.966,318.024,-145.227,170.161,51.539,160.042
C00620=1015.973,318.271,-145.261,170.168,51.535,160.043
C00621=1015.979,318.518,-145.294,170.174,51.531,160.043
C00622=1015.986,318.767,-145.327,170.181,51.526,160.043
C00623=1015.993,319.014,-145.360,170.187,51.521,160.043
C00624=1015.999,319.262,-145.394,170.194,51.517,160.043
C00625=1016.006,319.509,-145.427,170.200,51.512,160.043
C00626=1016.012,319.758,-145.460,170.207,51.508,160.043
C00627=1016.019,320.004,-145.494,170.213,51.503,160.043
C00628=1016.025,320.252,-145.527,170.220,51.499,160.044
C00629=1016.032,320.500,-145.561,170.226,51.494,160.044
C00630=1016.038,320.748,-145.594,170.233,51.489,160.044
C00631=1016.045,320.995,-145.628,170.239,51.485,160.044
C00632=1016.052,321.242,-145.661,170.246,51.480,160.044
C00633=1016.058,321.491,-145.695,170.253,51.476,160.045
C00634=1016.065,321.738,-145.728,170.259,51.472,160.045
C00635=1016.072,321.986,-145.761,170.266,51.467,160.045
C00636=1016.079,322.234,-145.795,170.273,51.463,160.045
C00637=1016.086,322.509,-145.833,170.280,51.458,160.045
C00638=1016.093,322.785,-145.870,170.288,51.452,160.045
C00639=1016.100,323.061,-145.908,170.294,51.448,160.045
C00640=1016.108,323.336,-145.944,170.303,51.443,160.046
C00641=1016.115,323.584,-145.979,170.309,51.438,160.046
C00642=1016.121,323.831,-146.012,170.316,51.434,160.046
C00643=1016.128,324.079,-146.046,170.322,51.429,160.046
C00644=1016.136,324.327,-146.080,170.330,51.425,160.046
C00645=1016.141,324.574,-146.113,170.335,51.421,160.046
C00646=1016.148,324.822,-146.147,170.343,51.416,160.047
C00647=1016.156,325.070,-146.181,170.350,51.412,160.047
C00648=1016.162,325.317,-146.214,170.356,51.408,160.047
C00649=1016.169,325.564,-146.248,170.363,51.404,160.047
C00650=1016.176,325.812,-146.283,170.370,51.399,160.048
C00651=1016.183,326.060,-146.316,170.377,51.395,160.048
C00652=1016.189,326.307,-146.350,170.383,51.391,160.048
C00653=1016.196,326.555,-146.384,170.390,51.386,160.048
C00654=1016.203,326.803,-146.419,170.396,51.383,160.049
C00655=1016.209,327.050,-146.453,170.403,51.378,160.049
C00656=1016.216,327.297,-146.487,170.411,51.374,160.049
C00657=1016.222,327.545,-146.522,170.417,51.370,160.049
C00658=1016.229,327.793,-146.556,170.424,51.366,160.050
C00659=1016.236,328.040,-146.590,170.431,51.362,160.050
C00660=1016.242,328.288,-146.625,170.437,51.358,160.050
C00661=1016.249,328.536,-146.659,170.445,51.354,160.051
C00662=1016.256,328.783,-146.694,170.452,51.350,160.051
C00663=1016.263,329.031,-146.728,170.458,51.346,160.051
C00664=1016.269,329.278,-146.763,170.465,51.342,160.051
C00665=1016.276,329.525,-146.797,170.472,51.337,160.052
C00666=1016.283,329.773,-146.831,170.479,51.334,160.052
C00667=1016.289,330.020,-146.866,170.486,51.329,160.052
C00668=1016.297,330.268,-146.900,170.493,51.325,160.053
C00669=1016.303,330.515,-146.935,170.499,51.321,160.053
C00670=1016.310,330.763,-146.970,170.507,51.318,160.053
C00671=1016.317,331.011,-147.004,170.514,51.314,160.054
C00672=1016.324,331.258,-147.039,170.520,51.310,160.054
C00673=1016.330,331.506,-147.074,170.527,51.306,160.054
C00674=1016.337,331.753,-147.109,170.535,51.301,160.054
C00675=1016.344,332.001,-147.143,170.541,51.298,160.055
C00676=1016.351,332.248,-147.178,170.548,51.294,160.055
C00677=1016.358,332.496,-147.213,170.556,51.290,160.056
C00678=1016.364,332.744,-147.247,170.562,51.287,160.056
C00679=1016.371,332.991,-147.283,170.569,51.282,160.056
C00680=1016.378,333.238,-147.318,170.577,51.278,160.057
C00681=1016.385,333.485,-147.352,170.583,51.275,160.057
C00682=1016.392,333.733,-147.387,170.590,51.271,160.057
C00683=1016.399,333.980,-147.422,170.598,51.267,160.058
C00684=1016.406,334.227,-147.458,170.604,51.263,160.058
C00685=1016.413,334.475,-147.493,170.612,51.260,160.059
C00686=1016.419,334.722,-147.528,170.619,51.256,160.059
C00687=1016.426,334.970,-147.563,170.627,51.252,160.059
C00688=1016.433,335.217,-147.598,170.633,51.248,160.060
C00689=1016.440,335.464,-147.633,170.640,51.245,160.060
C00690=1016.447,335.712,-147.669,170.648,51.241,160.060
C00691=1016.454,335.960,-147.704,170.654,51.237,160.061
C00692=1016.461,336.207,-147.739,170.662,51.234,160.061
C00693=1016.467,336.454,-147.774,170.669,51.230,160.062
C00694=1016.474,336.702,-147.809,170.676,51.226,160.062
C00695=1016.481,336.950,-147.845,170.683,51.223,160.063
C00696=1016.488,337.197,-147.880,170.690,51.219,160.063
C00697=1016.496,337.469,-147.919,170.698,51.215,160.063
C00698=1016.504,337.740,-147.958,170.706,51.211,160.064
C00699=1016.512,338.011,-147.997,170.714,51.207,160.064
C00700=1016.519,338.283,-148.035,170.722,51.203,160.065
C00701=1016.526,338.530,-148.071,170.730,51.199,160.065
C00702=1016.534,338.778,-148.106,170.736,51.196,160.066
C00703=1016.540,339.025,-148.141,170.744,51.192,160.066
C00704=1016.547,339.272,-148.177,170.751,51.189,160.067
C00705=1016.554,339.519,-148.212,170.759,51.185,160.067
C00706=1016.561,339.767,-148.249,170.766,51.182,160.068
C00707=1016.568,340.014,-148.284,170.773,51.178,160.068
C00708=1016.575,340.261,-148.320,170.781,51.175,160.069
C00709=1016.582,340.509,-148.355,170.787,51.172,160.069
C00710=1016.589,340.756,-148.391,170.795,51.168,160.070
C00711=1016.596,341.004,-148.428,170.803,51.165,160.070
C00712=1016.603,341.251,-148.463,170.810,51.161,160.071
C00713=1016.610,341.498,-148.499,170.817,51.158,160.071
C00714=1016.618,341.746,-148.535,170.824,51.154,160.072
C00715=1016.625,341.993,-148.570,170.832,51.151,160.072
C00716=1016.632,342.240,-148.607,170.840,51.147,160.073
C00717=1016.639,342.487,-148.643,170.847,51.145,160.073
C00718=1016.646,342.735,-148.679,170.854,51.141,160.074
C00719=1016.653,342.982,-148.714,170.862,51.138,160.074
C00720=1016.660,343.230,-148.751,170.869,51.134,160.075
C00721=1016.667,343.476,-148.787,170.876,51.131,160.075
C00722=1016.675,343.724,-148.823,170.884,51.128,160.076
C00723=1016.681,343.971,-148.860,170.892,51.125,160.076
C00724=1016.688,344.219,-148.895,170.899,51.121,160.077
C00725=1016.696,344.466,-148.932,170.907,51.118,160.078
C00726=1016.703,344.713,-148.967,170.914,51.115,160.078
C00727=1016.710,344.961,-149.004,170.921,51.111,160.079
C00728=1016.717,345.208,-149.040,170.929,51.109,160.079
C00729=1016.725,345.455,-149.076,170.937,51.105,160.080
C00730=1016.732,345.703,-149.113,170.945,51.102,160.081
C00731=1016.739,345.950,-149.149,170.952,51.099,160.081
C00732=1016.747,346.196,-149.186,170.959,51.095,160.082
C00733=1016.755,346.444,-149.222,170.967,51.092,160.082
C00734=1016.761,346.691,-149.259,170.975,51.089,160.083
C00735=1016.769,346.938,-149.295,170.983,51.086,160.083
C00736=1016.776,347.186,-149.332,170.991,51.083,160.084
C00737=1016.784,347.433,-149.368,170.997,51.080,160.085
C00738=1016.790,347.680,-149.405,171.005,51.077,160.085
C00739=1016.798,347.927,-149.441,171.013,51.074,160.086
C00740=1016.805,348.175,-149.479,171.021,51.071,160.087
C00741=1016.812,348.422,-149.515,171.029,51.068,160.087
C00742=1016.819,348.668,-149.552,171.037,51.065,160.088
C00743=1016.827,348.916,-149.588,171.044,51.062,160.088
C00744=1016.834,349.164,-149.625,171.052,51.059,160.089
C00745=1016.842,349.410,-149.662,171.060,51.056,160.090
C00746=1016.849,349.658,-149.699,171.068,51.053,160.091
C00747=1016.855,349.905,-149.736,171.075,51.049,160.091
C00748=1016.863,350.151,-149.773,171.083,51.047,160.092
C00749=1016.870,350.399,-149.810,171.091,51.044,160.093
C00750=1016.878,350.646,-149.847,171.098,51.041,160.093
C00751=1016.885,350.894,-149.883,171.106,51.038,160.094
C00752=1016.893,351.141,-149.920,171.114,51.035,160.095
C00753=1016.900,351.388,-149.958,171.122,51.032,160.095
C00754=1016.908,351.635,-149.994,171.130,51.030,160.096
C00755=1016.915,351.882,-150.032,171.138,51.027,160.097
C00756=1016.923,352.130,-150.069,171.146,51.024,160.097
C00757=1016.931,352.398,-150.109,171.154,51.021,160.098
C00758=1016.940,352.667,-150.150,171.163,51.018,160.099
C00759=1016.947,352.936,-150.190,171.172,51.014,160.100
C00760=1016.955,353.204,-150.230,171.180,51.011,160.101
C00761=1016.963,353.451,-150.267,171.188,51.009,160.101
C00762=1016.971,353.698,-150.305,171.196,51.006,160.102
C00763=1016.978,353.946,-150.342,171.204,51.003,160.103
C00764=1016.985,354.193,-150.380,171.213,51.001,160.104
C00765=1016.993,354.440,-150.417,171.221,50.998,160.104
C00766=1017.000,354.687,-150.454,171.229,50.995,160.105
C00767=1017.008,354.934,-150.492,171.237,50.992,160.106
C00768=1017.015,355.180,-150.530,171.245,50.990,160.107
C00769=1017.023,355.427,-150.567,171.253,50.987,160.107
C00770=1017.030,355.674,-150.605,171.261,50.984,160.108
C00771=1017.038,355.922,-150.643,171.269,50.982,160.109
C00772=1017.046,356.169,-150.680,171.277,50.979,160.110
C00773=1017.054,356.415,-150.718,171.285,50.976,160.110
C00774=1017.061,356.663,-150.755,171.294,50.973,160.111
C00775=1017.068,356.910,-150.793,171.302,50.971,160.112
C00776=1017.076,357.158,-150.831,171.310,50.968,160.113
C00777=1017.084,357.404,-150.868,171.318,50.965,160.114
C00778=1017.092,357.651,-150.906,171.327,50.963,160.115
C00779=1017.100,357.898,-150.944,171.335,50.960,160.115
C00780=1017.107,358.145,-150.982,171.343,50.958,160.116
C00781=1017.115,358.392,-151.020,171.351,50.955,160.117
C00782=1017.122,358.640,-151.058,171.359,50.953,160.118
C00783=1017.131,358.886,-151.096,171.368,50.951,160.119
C00784=1017.138,359.133,-151.133,171.376,50.948,160.120
C00785=1017.146,359.380,-151.172,171.384,50.945,160.121
C00786=1017.154,359.627,-151.210,171.393,50.943,160.121
C00787=1017.161,359.874,-151.248,171.401,50.941,160.122
C00788=1017.168,360.121,-151.287,171.409,50.938,160.123
C00789=1017.176,360.368,-151.325,171.417,50.936,160.124
C00790=1017.183,360.614,-151.363,171.426,50.933,160.125
C00791=1017.192,360.862,-151.402,171.434,50.931,160.126
C00792=1017.199,361.108,-151.440,171.443,50.929,160.127
C00793=1017.207,361.356,-151.478,171.451,50.927,160.128
C00794=1017.215,361.602,-151.516,171.459,50.924,160.129
C00795=1017.223,361.850,-151.555,171.468,50.922,160.130
C00796=1017.230,362.096,-151.593,171.476,50.920,160.130
C00797=1017.238,362.343,-151.632,171.485,50.918,160.131
C00798=1017.246,362.590,-151.670,171.494,50.915,160.132
C00799=1017.254,362.837,-151.709,171.502,50.913,160.133
C00800=1017.261,363.084,-151.748,171.511,50.910,160.134
C00801=1017.269,363.331,-151.787,171.519,50.908,160.135
C00802=1017.278,363.578,-151.825,171.528,50.906,160.136
C00803=1017.285,363.824,-151.864,171.536,50.904,160.137
C00804=1017.293,364.071,-151.902,171.544,50.901,160.138
C00805=1017.301,364.319,-151.941,171.553,50.899,160.139
C00806=1017.309,364.565,-151.979,171.563,50.897,160.140
C00807=1017.317,364.812,-152.018,171.571,50.895,160.141
C00808=1017.326,365.059,-152.057,171.579,50.892,160.142
C00809=1017.333,365.306,-152.095,171.588,50.890,160.143
C00810=1017.342,365.552,-152.135,171.597,50.889,160.144
C00811=1017.350,365.799,-152.173,171.606,50.886,160.145
C00812=1017.357,366.047,-152.212,171.614,50.884,160.146
C00813=1017.365,366.293,-152.251,171.623,50.881,160.147
C00814=1017.373,366.540,-152.290,171.632,50.880,160.148
C00815=1017.382,366.787,-152.329,171.640,50.877,160.149
C00816=1017.390,367.034,-152.368,171.650,50.875,160.150
C00817=1017.399,367.310,-152.412,171.659,50.873,160.151
C00818=1017.408,367.586,-152.456,171.669,50.871,160.152
C00819=1017.417,367.862,-152.500,171.679,50.869,160.154
C00820=1017.425,368.138,-152.544,171.690,50.866,160.155
C00821=1017.434,368.385,-152.583,171.698,50.864,160.156
C00822=1017.442,368.632,-152.622,171.707,50.863,160.157
C00823=1017.450,368.879,-152.662,171.716,50.861,160.158
C00824=1017.458,369.125,-152.701,171.725,50.858,160.159
C00825=1017.466,369.372,-152.741,171.734,50.857,160.160
C00826=1017.474,369.618,-152.780,171.742,50.855,160.161
C00827=1017.482,369.865,-152.819,171.751,50.853,160.162
C00828=1017.490,370.112,-152.859,171.761,50.851,160.163
C00829=1017.498,370.358,-152.899,171.769,50.849,160.165
C00830=1017.506,370.605,-152.939,171.778,50.847,160.166
C00831=1017.515,370.852,-152.978,171.788,50.845,160.167
C00832=1017.522,371.099,-153.018,171.797,50.844,160.168
C00833=1017.531,371.346,-153.058,171.806,50.842,160.169
C00834=1017.540,371.593,-153.097,171.815,50.839,160.170
C00835=1017.548,371.840,-153.137,171.824,50.838,160.171
C00836=1017.556,372.086,-153.177,171.833,50.836,160.172
C00837=1017.564,372.332,-153.217,171.842,50.834,160.174
C00838=1017.573,372.579,-153.256,171.851,50.832,160.175
C00839=1017.581,372.826,-153.295,171.861,50.831,160.176
C00840=1017.589,373.072,-153.336,171.870,50.829,160.177
C00841=1017.598,373.319,-153.376,171.879,50.828,160.179
C00842=1017.606,373.566,-153.416,171.889,50.826,160.180
C00843=1017.615,373.812,-153.456,171.898,50.824,160.181
C00844=1017.622,374.059,-153.496,171.907,50.822,160.182
C00845=1017.632,374.306,-153.536,171.916,50.820,160.183
C00846=1017.640,374.552,-153.575,171.926,50.819,160.185
C00847=1017.648,374.799,-153.616,171.935,50.817,160.186
C00848=1017.657,375.045,-153.655,171.945,50.815,160.187
C00849=1017.665,375.292,-153.696,171.954,50.814,160.188
C00850=1017.674,375.538,-153.736,171.964,50.812,160.190
C00851=1017.682,375.786,-153.777,171.973,50.810,160.191
C00852=1017.691,376.032,-153.817,171.982,50.808,160.192
C00853=1017.699,376.278,-153.857,171.992,50.807,160.193
C00854=1017.708,376.525,-153.898,172.000,50.806,160.194
C00855=1017.716,376.771,-153.939,172.011,50.804,160.196
C00856=1017.725,377.017,-153.979,172.020,50.803,160.197
C00857=1017.733,377.264,-154.020,172.030,50.801,160.198
C00858=1017.741,377.510,-154.061,172.040,50.800,160.200
C00859=1017.750,377.757,-154.102,172.049,50.798,160.201
C00860=1017.758,378.004,-154.142,172.059,50.797,160.202
C00861=1017.767,378.250,-154.183,172.068,50.796,160.204
C00862=1017.775,378.497,-154.223,172.078,50.794,160.205
C00863=1017.784,378.744,-154.264,172.087,50.793,160.206
C00864=1017.792,378.990,-154.305,172.097,50.791,160.208
C00865=1017.801,379.237,-154.345,172.107,50.790,160.209
C00866=1017.810,379.482,-154.387,172.116,50.789,160.210
C00867=1017.818,379.729,-154.428,172.126,50.787,160.212
C00868=1017.827,379.976,-154.469,172.135,50.786,160.213
C00869=1017.836,380.222,-154.509,172.146,50.784,160.214
C00870=1017.845,380.469,-154.550,172.156,50.783,160.216
C00871=1017.853,380.715,-154.591,172.165,50.782,160.217
C00872=1017.861,380.961,-154.633,172.175,50.780,160.219
C00873=1017.871,381.208,-154.673,172.185,50.779,160.220
C00874=1017.880,381.454,-154.715,172.194,50.778,160.221
C00875=1017.888,381.701,-154.756,172.205,50.776,160.223
C00876=1017.897,381.947,-154.797,172.215,50.775,160.224
C00877=1017.907,382.246,-154.847,172.226,50.774,160.226
C00878=1017.918,382.545,-154.897,172.239,50.772,160.228
C00879=1017.929,382.843,-154.947,172.251,50.770,160.229
C00880=1017.940,383.142,-154.996,172.263,50.769,160.231
C00881=1017.949,383.388,-155.038,172.273,50.768,160.233
C00882=1017.958,383.634,-155.079,172.283,50.767,160.234
C00883=1017.967,383.880,-155.121,172.294,50.765,160.236
C00884=1017.976,384.127,-155.162,172.303,50.764,160.237
C00885=1017.985,384.374,-155.204,172.313,50.763,160.239
C00886=1017.994,384.620,-155.245,172.324,50.762,160.240
C00887=1018.003,384.866,-155.286,172.334,50.760,160.241
C00888=1018.012,385.113,-155.328,172.344,50.760,160.243
C00889=1018.021,385.359,-155.370,172.355,50.758,160.244
C00890=1018.030,385.605,-155.412,172.365,50.757,160.246
C00891=1018.039,385.852,-155.453,172.374,50.756,160.247
C00892=1018.048,386.098,-155.495,172.385,50.756,160.249
C00893=1018.057,386.344,-155.538,172.395,50.755,160.251
C00894=1018.066,386.590,-155.579,172.406,50.753,160.252
C00895=1018.075,386.836,-155.621,172.416,50.752,160.254
C00896=1018.084,387.083,-155.663,172.427,50.752,160.255
C00897=1018.093,387.329,-155.705,172.437,50.750,160.257
C00898=1018.102,387.575,-155.747,172.447,50.749,160.259
C00899=1018.112,387.821,-155.790,172.458,50.748,160.260
C00900=1018.121,388.068,-155.831,172.469,50.748,160.262
C00901=1018.130,388.313,-155.874,172.479,50.747,160.263
C00902=1018.138,388.560,-155.916,172.490,50.746,160.265
C00903=1018.148,388.806,-155.958,172.500,50.745,160.267
C00904=1018.157,389.053,-156.001,172.511,50.744,160.268
C00905=1018.166,389.299,-156.043,172.521,50.743,160.270
C00906=1018.176,389.544,-156.085,172.532,50.742,160.271
C00907=1018.184,389.791,-156.128,172.543,50.742,160.273
C00908=1018.194,390.038,-156.171,172.553,50.741,160.275
C00909=1018.203,390.283,-156.213,172.564,50.740,160.277
C00910=1018.212,390.529,-156.255,172.574,50.739,160.278
C00911=1018.222,390.776,-156.298,172.585,50.738,160.280
C00912=1018.231,391.021,-156.341,172.596,50.737,160.281
C00913=1018.240,391.268,-156.384,172.606,50.737,160.283
C00914=1018.250,391.514,-156.426,172.617,50.736,160.285
C00915=1018.259,391.760,-156.469,172.629,50.735,160.287
C00916=1018.269,392.006,-156.512,172.639,50.734,160.288
C00917=1018.278,392.252,-156.554,172.650,50.734,160.290
C00918=1018.287,392.498,-156.598,172.661,50.733,160.292
C00919=1018.296,392.744,-156.640,172.672,50.733,160.294
C00920=1018.306,392.991,-156.683,172.682,50.732,160.295
C00921=1018.315,393.236,-156.726,172.694,50.731,160.297
C00922=1018.325,393.483,-156.769,172.705,50.731,160.299
C00923=1018.335,393.729,-156.812,172.716,50.730,160.301
C00924=1018.343,393.974,-156.856,172.726,50.729,160.302
C00925=1018.353,394.221,-156.899,172.738,50.729,160.304
C00926=1018.363,394.466,-156.942,172.749,50.728,160.306
C00927=1018.372,394.713,-156.985,172.760,50.728,160.308
C00928=1018.382,394.959,-157.029,172.772,50.727,160.310
C00929=1018.391,395.204,-157.071,172.783,50.727,160.312
C00930=1018.401,395.450,-157.115,172.793,50.726,160.313
C00931=1018.411,395.696,-157.159,172.805,50.725,160.315
C00932=1018.421,395.943,-157.202,172.816,50.725,160.317
C00933=1018.430,396.189,-157.246,172.827,50.725,160.319
C00934=1018.440,396.434,-157.289,172.839,50.724,160.321
C00935=1018.449,396.680,-157.333,172.850,50.724,160.323
C00936=1018.459,396.927,-157.376,172.861,50.724,160.325
C00937=1018.472,397.263,-157.436,172.877,50.723,160.327
C00938=1018.486,397.599,-157.496,172.893,50.723,160.330
C00939=1018.499,397.935,-157.556,172.908,50.722,160.332
C00940=1018.512,398.271,-157.616,172.924,50.721,160.335
C00941=1018.522,398.517,-157.659,172.936,50.721,160.337
C00942=1018.532,398.763,-157.703,172.947,50.720,160.339
C00943=1018.542,399.009,-157.747,172.959,50.720,160.341
C00944=1018.551,399.255,-157.791,172.970,50.720,160.343
C00945=1018.561,399.501,-157.836,172.982,50.719,160.345
C00946=1018.571,399.747,-157.879,172.993,50.719,160.347
C00947=1018.581,399.992,-157.924,173.006,50.719,160.349
C00948=1018.591,400.239,-157.968,173.018,50.718,160.351
C00949=1018.601,400.485,-158.012,173.029,50.719,160.353
C00950=1018.611,400.730,-158.057,173.041,50.718,160.355
C00951=1018.621,400.976,-158.101,173.052,50.718,160.357
C00952=1018.630,401.222,-158.145,173.065,50.718,160.359
C00953=1018.640,401.467,-158.190,173.077,50.718,160.361
C00954=1018.650,401.713,-158.235,173.088,50.718,160.363
C00955=1018.661,401.959,-158.279,173.100,50.718,160.365
C00956=1018.670,402.205,-158.323,173.112,50.717,160.367
C00957=1018.680,402.450,-158.368,173.124,50.717,160.369
C00958=1018.690,402.696,-158.413,173.136,50.717,160.371
C00959=1018.701,402.942,-158.458,173.148,50.717,160.373
C00960=1018.711,403.187,-158.502,173.161,50.717,160.376
C00961=1018.720,403.433,-158.547,173.172,50.718,160.378
C00962=1018.731,403.679,-158.592,173.184,50.717,160.380
C00963=1018.741,403.924,-158.637,173.197,50.717,160.382
C00964=1018.751,404.170,-158.682,173.209,50.717,160.384
C00965=1018.761,404.416,-158.727,173.221,50.717,160.386
C00966=1018.771,404.661,-158.772,173.234,50.717,160.388
C00967=1018.782,404.907,-158.816,173.245,50.717,160.390
C00968=1018.792,405.153,-158.862,173.258,50.717,160.393
C00969=1018.802,405.398,-158.907,173.270,50.717,160.395
C00970=1018.812,405.645,-158.952,173.283,50.718,160.397
C00971=1018.823,405.889,-158.997,173.295,50.717,160.399
C00972=1018.834,406.135,-159.042,173.307,50.717,160.401
C00973=1018.844,406.382,-159.087,173.320,50.717,160.404
C00974=1018.855,406.626,-159.132,173.332,50.718,160.406
C00975=1018.865,406.872,-159.178,173.345,50.718,160.408
C00976=1018.876,407.118,-159.223,173.358,50.718,160.410
C00977=1018.885,407.364,-159.268,173.370,50.718,160.413
C00978=1018.897,407.609,-159.314,173.383,50.718,160.415
C00979=1018.907,407.854,-159.359,173.396,50.718,160.417
C00980=1018.918,408.101,-159.405,173.409,50.718,160.420
C00981=1018.928,408.346,-159.451,173.422,50.719,160.422
C00982=1018.939,408.592,-159.496,173.434,50.719,160.424
C00983=1018.950,408.837,-159.542,173.447,50.719,160.426
C00984=1018.960,409.083,-159.588,173.459,50.720,160.429
C00985=1018.970,409.328,-159.634,173.472,50.720,160.431
C00986=1018.981,409.573,-159.680,173.485,50.720,160.433
C00987=1018.991,409.819,-159.726,173.498,50.720,160.436
C00988=1019.002,410.065,-159.772,173.511,50.720,160.438
C00989=1019.013,410.310,-159.817,173.524,50.721,160.441
C00990=1019.024,410.555,-159.864,173.537,50.721,160.443
C00991=1019.034,410.801,-159.910,173.550,50.721,160.445
C00992=1019.045,411.046,-159.956,173.563,50.722,160.448
C00993=1019.055,411.292,-160.002,173.577,50.723,160.450
C00994=1019.067,411.538,-160.049,173.590,50.723,160.453
C00995=1019.078,411.783,-160.095,173.603,50.723,160.455
C00996=1019.088,412.028,-160.141,173.616,50.723,160.458
C00997=1019.104,412.387,-160.209,173.636,50.724,160.461
C00998=1019.120,412.745,-160.277,173.655,50.725,160.465
C00999=1019.136,413.104,-160.345,173.674,50.726,160.469
C01000=1019.152,413.462,-160.413,173.695,50.727,160.472
C01001=1019.164,413.708,-160.460,173.707,50.727,160.475
C01002=1019.175,413.953,-160.506,173.722,50.728,160.477
C01003=1019.185,414.198,-160.553,173.734,50.728,160.480
C01004=1019.196,414.444,-160.600,173.748,50.729,160.482
C01005=1019.207,414.689,-160.646,173.763,50.729,160.485
C01006=1019.218,414.935,-160.693,173.776,50.730,160.488
C01007=1019.229,415.180,-160.740,173.789,50.730,160.490
C01008=1019.240,415.425,-160.788,173.804,50.731,160.493
C01009=1019.255,415.744,-160.849,173.821,50.733,160.496
C01010=1019.269,416.063,-160.910,173.839,50.733,160.500
C01011=1019.284,416.381,-160.972,173.857,50.734,160.503
C01012=1019.298,416.700,-161.033,173.875,50.735,160.507
C01013=1019.309,416.946,-161.080,173.889,50.736,160.509
C01014=1019.321,417.191,-161.128,173.903,50.736,160.512
C01015=1019.332,417.436,-161.176,173.917,50.737,160.515
C01016=1019.343,417.681,-161.223,173.932,50.738,160.518
C01017=1019.355,417.926,-161.271,173.945,50.739,160.520
C01018=1019.367,418.172,-161.318,173.959,50.740,160.523
C01019=1019.377,418.417,-161.366,173.974,50.741,160.526
C01020=1019.389,418.662,-161.413,173.988,50.741,160.528
C01021=1019.018,416.680,-161.369,173.860,50.805,160.524
C01022=1019.006,416.435,-161.321,173.846,50.805,160.521
C01023=1018.995,416.190,-161.274,173.832,50.804,160.519
C01024=1018.984,415.944,-161.227,173.819,50.803,160.516
C01025=1018.973,415.700,-161.179,173.805,50.802,160.513
C01026=1018.962,415.454,-161.132,173.791,50.802,160.511
C01027=1018.951,415.209,-161.085,173.776,50.801,160.508
C01028=1018.940,414.963,-161.038,173.764,50.801,160.506
C01029=1018.929,414.718,-160.991,173.750,50.800,160.503
C01030=1018.917,414.473,-160.944,173.735,50.800,160.500
C01031=1018.907,414.228,-160.898,173.722,50.800,160.498
C01032=1018.895,413.982,-160.851,173.709,50.799,160.495
C01033=1018.884,413.737,-160.804,173.695,50.799,160.493
C01034=1018.866,413.334,-160.728,173.673,50.798,160.489
C01035=1018.848,412.930,-160.651,173.650,50.797,160.484
C01036=1018.830,412.527,-160.575,173.629,50.797,160.480
C01037=1018.812,412.123,-160.499,173.607,50.796,160.476
C01038=1018.802,411.877,-160.452,173.593,50.796,160.474
C01039=1018.791,411.632,-160.406,173.580,50.795,160.471
C01040=1018.781,411.387,-160.360,173.567,50.795,160.469
C01041=1018.770,411.142,-160.313,173.554,50.795,160.467
C01042=1018.759,410.896,-160.267,173.541,50.795,160.464
C01043=1018.748,410.651,-160.221,173.527,50.795,160.462
C01044=1018.738,410.405,-160.175,173.515,50.794,160.459
C01045=1018.727,410.160,-160.129,173.501,50.794,160.457
C01046=1018.716,409.914,-160.083,173.488,50.794,160.455
C01047=1018.706,409.669,-160.037,173.475,50.793,160.452
C01048=1018.695,409.423,-159.991,173.463,50.793,160.450
C01049=1018.684,409.178,-159.945,173.449,50.793,160.448
C01050=1018.674,408.932,-159.899,173.436,50.793,160.445
C01051=1018.663,408.686,-159.853,173.424,50.792,160.443
C01052=1018.652,408.441,-159.807,173.411,50.793,160.441
C01053=1018.642,408.195,-159.762,173.398,50.792,160.438
C01054=1018.632,407.955,-159.717,173.385,50.793,160.436
C01055=1018.621,407.715,-159.673,173.372,50.792,160.434
C01056=1018.611,407.474,-159.629,173.360,50.792,160.431
C01057=1018.600,407.234,-159.585,173.349,50.792,160.429
C01058=1018.591,406.994,-159.540,173.336,50.792,160.427
C01059=1018.580,406.754,-159.495,173.324,50.792,160.425
C01060=1018.569,406.514,-159.451,173.311,50.792,160.423
C01061=1018.560,406.274,-159.407,173.299,50.792,160.421
C01062=1018.549,406.027,-159.362,173.287,50.792,160.418
C01063=1018.539,405.782,-159.318,173.274,50.792,160.416
C01064=1018.528,405.536,-159.272,173.262,50.792,160.414
C01065=1018.519,405.291,-159.227,173.249,50.792,160.412
C01066=1018.508,405.045,-159.182,173.237,50.793,160.410
C01067=1018.498,404.800,-159.137,173.225,50.793,160.408
C01068=1018.487,404.554,-159.091,173.212,50.793,160.405
C01069=1018.477,404.308,-159.047,173.200,50.793,160.403
C01070=1018.466,404.063,-159.002,173.188,50.793,160.401
C01071=1018.457,403.817,-158.957,173.175,50.793,160.399
C01072=1018.447,403.572,-158.912,173.163,50.793,160.397
C01073=1018.437,403.325,-158.867,173.151,50.793,160.395
C01074=1018.426,403.080,-158.823,173.138,50.793,160.392
C01075=1018.417,402.835,-158.778,173.127,50.794,160.391
C01076=1018.406,402.588,-158.733,173.115,50.794,160.388
C01077=1018.397,402.342,-158.689,173.102,50.794,160.386
C01078=1018.386,402.097,-158.645,173.091,50.795,160.384
C01079=1018.376,401.851,-158.599,173.078,50.795,160.382
C01080=1018.366,401.605,-158.555,173.067,50.794,160.380
C01081=1018.356,401.359,-158.511,173.055,50.795,160.378
C01082=1018.346,401.114,-158.466,173.042,50.795,160.376
C01083=1018.337,400.868,-158.421,173.031,50.796,160.374
C01084=1018.327,400.622,-158.377,173.019,50.796,160.372
C01085=1018.317,400.377,-158.333,173.007,50.796,160.370
C01086=1018.307,400.131,-158.289,172.995,50.797,160.368
C01087=1018.297,399.884,-158.245,172.984,50.797,160.366
C01088=1018.287,399.639,-158.200,172.972,50.797,160.364
C01089=1018.278,399.393,-158.156,172.960,50.798,160.362
C01090=1018.267,399.147,-158.113,172.949,50.798,160.360
C01091=1018.258,398.901,-158.068,172.937,50.798,160.358
C01092=1018.248,398.656,-158.024,172.926,50.799,160.356
C01093=1018.238,398.410,-157.980,172.914,50.799,160.354
C01094=1018.225,398.060,-157.919,172.897,50.800,160.352
C01095=1018.211,397.711,-157.856,172.881,50.801,160.349
C01096=1018.197,397.361,-157.794,172.864,50.802,160.346
C01097=1018.183,397.012,-157.732,172.849,50.802,160.344
C01098=1018.173,396.766,-157.688,172.837,50.803,160.342
C01099=1018.163,396.520,-157.645,172.826,50.803,160.340
C01100=1018.155,396.274,-157.601,172.814,50.804,160.338
C01101=1018.144,396.028,-157.558,172.803,50.805,160.336
C01102=1018.135,395.782,-157.515,172.791,50.806,160.334
C01103=1018.125,395.536,-157.471,172.780,50.806,160.332
C01104=1018.116,395.291,-157.428,172.769,50.806,160.331
C01105=1018.106,395.044,-157.385,172.758,50.807,160.329
C01106=1018.096,394.798,-157.341,172.747,50.808,160.327
C01107=1018.087,394.552,-157.298,172.735,50.809,160.325
C01108=1018.077,394.306,-157.255,172.724,50.809,160.323
C01109=1018.068,394.060,-157.211,172.714,50.810,160.322
C01110=1018.059,393.814,-157.169,172.702,50.811,160.320
C01111=1018.049,393.568,-157.125,172.691,50.812,160.318
C01112=1018.040,393.322,-157.082,172.680,50.812,160.316
C01113=1018.030,393.076,-157.040,172.668,50.813,160.315
C01114=1018.021,392.830,-156.996,172.658,50.814,160.313
C01115=1018.012,392.584,-156.953,172.647,50.814,160.311
C01116=1018.002,392.338,-156.911,172.636,50.815,160.309
C01117=1017.992,392.092,-156.868,172.625,50.816,160.308
C01118=1017.983,391.846,-156.825,172.614,50.817,160.306
C01119=1017.974,391.599,-156.782,172.603,50.817,160.304
C01120=1017.965,391.353,-156.739,172.593,50.818,160.302
C01121=1017.955,391.107,-156.697,172.582,50.819,160.301
C01122=1017.946,390.861,-156.654,172.570,50.820,160.299
C01123=1017.937,390.615,-156.612,172.560,50.821,160.297
C01124=1017.927,390.369,-156.569,172.549,50.822,160.296
C01125=1017.918,390.123,-156.526,172.539,50.823,160.294
C01126=1017.909,389.877,-156.484,172.528,50.824,160.293
C01127=1017.899,389.630,-156.441,172.518,50.825,160.291
C01128=1017.890,389.384,-156.399,172.506,50.826,160.289
C01129=1017.881,389.138,-156.357,172.495,50.827,160.288
C01130=1017.872,388.892,-156.315,172.485,50.828,160.286
C01131=1017.863,388.645,-156.272,172.474,50.828,160.284
C01132=1017.854,388.399,-156.230,172.464,50.830,160.283
C01133=1017.845,388.153,-156.187,172.454,50.831,160.281
C01134=1017.836,387.907,-156.146,172.443,50.832,160.280
C01135=1017.827,387.661,-156.103,172.433,50.833,160.278
C01136=1017.818,387.415,-156.062,172.422,50.834,160.276
C01137=1017.808,387.168,-156.019,172.412,50.835,160.275
C01138=1017.799,386.921,-155.978,172.401,50.836,160.273
C01139=1017.790,386.676,-155.935,172.391,50.837,160.272
C01140=1017.781,386.429,-155.894,172.381,50.839,160.270
C01141=1017.772,386.183,-155.852,172.370,50.839,160.269
C01142=1017.763,385.937,-155.810,172.360,50.841,160.267
C01143=1017.754,385.690,-155.768,172.349,50.842,160.266
C01144=1017.745,385.445,-155.726,172.339,50.843,160.264
C01145=1017.736,385.198,-155.684,172.329,50.844,160.262
C01146=1017.727,384.952,-155.643,172.318,50.845,160.261
C01147=1017.718,384.705,-155.601,172.308,50.847,160.260
C01148=1017.710,384.458,-155.560,172.298,50.848,160.258
C01149=1017.700,384.212,-155.519,172.287,50.849,160.257
C01150=1017.691,383.966,-155.477,172.277,50.851,160.255
C01151=1017.682,383.720,-155.435,172.268,50.852,160.254
C01152=1017.674,383.473,-155.395,172.258,50.853,160.252
C01153=1017.664,383.227,-155.354,172.248,50.855,160.251
C01154=1017.653,382.927,-155.303,172.235,50.856,160.249
C01155=1017.642,382.625,-155.253,172.223,50.858,160.247
C01156=1017.631,382.324,-155.202,172.210,50.859,160.245
C01157=1017.621,382.023,-155.152,172.199,50.861,160.244
C01158=1017.612,381.777,-155.110,172.189,50.863,160.242
C01159=1017.604,381.531,-155.070,172.178,50.864,160.241
C01160=1017.594,381.284,-155.028,172.168,50.865,160.240
C01161=1017.586,381.037,-154.987,172.158,50.867,160.238
C01162=1017.577,380.792,-154.946,172.149,50.868,160.237
C01163=1017.569,380.545,-154.905,172.139,50.869,160.235
C01164=1017.559,380.298,-154.865,172.129,50.871,160.234
C01165=1017.551,380.052,-154.823,172.119,50.873,160.233
C01166=1017.542,379.806,-154.782,172.110,50.874,160.231
C01167=1017.534,379.559,-154.742,172.099,50.875,160.230
C01168=1017.526,379.312,-154.701,172.090,50.877,160.229
C01169=1017.516,379.066,-154.660,172.080,50.878,160.227
C01170=1017.508,378.820,-154.619,172.070,50.880,160.226
C01171=1017.499,378.573,-154.578,172.060,50.882,160.225
C01172=1017.491,378.327,-154.537,172.051,50.883,160.223
C01173=1017.482,378.080,-154.497,172.041,50.885,160.222
C01174=1017.474,377.834,-154.456,172.031,50.886,160.221
C01175=1017.466,377.587,-154.416,172.022,50.888,160.220
C01176=1017.457,377.340,-154.375,172.012,50.890,160.218
C01177=1017.448,377.094,-154.335,172.003,50.891,160.217
C01178=1017.440,376.847,-154.294,171.993,50.893,160.216
C01179=1017.432,376.601,-154.253,171.983,50.895,160.214
C01180=1017.424,376.355,-154.212,171.974,50.896,160.213
C01181=1017.414,376.108,-154.172,171.965,50.898,160.212
C01182=1017.407,375.861,-154.132,171.956,50.899,160.211
C01183=1017.399,375.615,-154.091,171.946,50.901,160.209
C01184=1017.389,375.368,-154.051,171.937,50.903,160.208
C01185=1017.382,375.121,-154.011,171.927,50.905,160.207
C01186=1017.373,374.875,-153.971,171.917,50.907,160.206
C01187=1017.364,374.628,-153.931,171.908,50.908,160.205
C01188=1017.356,374.382,-153.891,171.899,50.910,160.203
C01189=1017.347,374.135,-153.851,171.889,50.911,160.202
C01190=1017.339,373.889,-153.811,171.880,50.913,160.201
C01191=1017.330,373.642,-153.771,171.871,50.915,160.200
C01192=1017.322,373.395,-153.731,171.861,50.917,160.198
C01193=1017.314,373.149,-153.691,171.852,50.919,160.197
C01194=1017.305,372.902,-153.652,171.842,50.921,160.196
C01195=1017.298,372.655,-153.612,171.834,50.923,160.195
C01196=1017.288,372.409,-153.571,171.824,50.925,160.194
C01197=1017.280,372.162,-153.531,171.815,50.927,160.193
C01198=1017.272,371.915,-153.492,171.806,50.929,160.192
C01199=1017.264,371.669,-153.453,171.797,50.931,160.190
C01200=1017.256,371.422,-153.413,171.787,50.933,160.189
C01201=1017.247,371.175,-153.374,171.778,50.934,160.188
C01202=1017.240,370.928,-153.334,171.770,50.937,160.187
C01203=1017.231,370.682,-153.294,171.760,50.939,160.186
C01204=1017.223,370.435,-153.255,171.751,50.940,160.185
C01205=1017.215,370.188,-153.215,171.742,50.942,160.183
C01206=1017.207,369.941,-153.176,171.733,50.945,160.183
C01207=1017.199,369.695,-153.136,171.724,50.946,160.181
C01208=1017.190,369.448,-153.097,171.715,50.948,160.180
C01209=1017.183,369.201,-153.057,171.706,50.951,160.179
C01210=1017.174,368.954,-153.017,171.697,50.952,160.178
C01211=1017.166,368.709,-152.978,171.688,50.955,160.177
C01212=1017.159,368.462,-152.938,171.679,50.957,160.176
C01213=1017.150,368.214,-152.900,171.671,50.959,160.175
C01214=1017.142,367.936,-152.855,171.660,50.961,160.174
C01215=1017.133,367.657,-152.810,171.650,50.963,160.173
C01216=1017.123,367.379,-152.766,171.640,50.966,160.171
C01217=1017.114,367.100,-152.722,171.630,50.968,160.170
C01218=1017.107,366.854,-152.683,171.622,50.971,160.169
C01219=1017.098,366.607,-152.644,171.612,50.973,160.168
C01220=1017.090,366.360,-152.605,171.603,50.975,160.167
C01221=1017.082,366.113,-152.567,171.595,50.977,160.166
C01222=1017.074,365.866,-152.528,171.586,50.980,160.165
C01223=1017.066,365.620,-152.489,171.577,50.982,160.164
C01224=1017.058,365.373,-152.450,171.568,50.984,160.163
C01225=1017.050,365.126,-152.412,171.560,50.986,160.162
C01226=1017.042,364.880,-152.373,171.551,50.989,160.161
C01227=1017.033,364.632,-152.334,171.542,50.991,160.160
C01228=1017.025,364.385,-152.296,171.534,50.993,160.159
C01229=1017.018,364.139,-152.257,171.525,50.996,160.158
C01230=1017.010,363.891,-152.218,171.516,50.998,160.157
C01231=1017.002,363.645,-152.179,171.508,51.000,160.156
C01232=1016.994,363.398,-152.141,171.499,51.003,160.156
C01233=1016.986,363.151,-152.102,171.491,51.005,160.155
C01234=1016.979,362.904,-152.064,171.481,51.008,160.154
C01235=1016.971,362.657,-152.025,171.473,51.010,160.153
C01236=1016.963,362.411,-151.987,171.465,51.012,160.152
C01237=1016.955,362.163,-151.948,171.456,51.015,160.151
C01238=1016.947,361.917,-151.910,171.448,51.017,160.150
C01239=1016.939,361.670,-151.871,171.440,51.020,160.149
C01240=1016.932,361.423,-151.833,171.430,51.022,160.148
C01241=1016.924,361.175,-151.795,171.422,51.025,160.147
C01242=1016.916,360.929,-151.757,171.414,51.027,160.146
C01243=1016.909,360.681,-151.718,171.405,51.029,160.145
C01244=1016.901,360.435,-151.680,171.397,51.032,160.145
C01245=1016.894,360.188,-151.641,171.389,51.034,160.144
C01246=1016.886,359.940,-151.603,171.380,51.037,160.143
C01247=1016.878,359.694,-151.565,171.372,51.040,160.142
C01248=1016.871,359.447,-151.527,171.363,51.042,160.141
C01249=1016.863,359.200,-151.488,171.355,51.045,160.140
C01250=1016.855,358.953,-151.451,171.347,51.047,160.139
C01251=1016.848,358.707,-151.413,171.338,51.050,160.138
C01252=1016.840,358.459,-151.375,171.330,51.053,160.138
C01253=1016.832,358.212,-151.337,171.322,51.055,160.137
C01254=1016.824,357.965,-151.299,171.314,51.058,160.136
C01255=1016.817,357.717,-151.262,171.305,51.060,160.135
C01256=1016.809,357.471,-151.223,171.297,51.063,160.134
C01257=1016.802,357.224,-151.186,171.288,51.066,160.134
C01258=1016.794,356.977,-151.149,171.280,51.069,160.133
C01259=1016.786,356.730,-151.110,171.272,51.071,160.132
C01260=1016.778,356.483,-151.073,171.264,51.074,160.131
C01261=1016.771,356.236,-151.035,171.256,51.077,160.130
C01262=1016.763,355.989,-150.998,171.248,51.080,160.130
C01263=1016.756,355.742,-150.960,171.240,51.082,160.129
C01264=1016.748,355.495,-150.923,171.232,51.085,160.128
C01265=1016.741,355.247,-150.885,171.223,51.088,160.127
C01266=1016.733,355.000,-150.848,171.215,51.091,160.127
C01267=1016.725,354.753,-150.810,171.207,51.094,160.126
C01268=1016.718,354.506,-150.773,171.199,51.096,160.125
C01269=1016.711,354.259,-150.735,171.191,51.099,160.124
C01270=1016.703,354.012,-150.698,171.183,51.102,160.124
C01271=1016.696,353.765,-150.661,171.175,51.105,160.123
C01272=1016.688,353.518,-150.623,171.167,51.107,160.122
C01273=1016.681,353.271,-150.586,171.159,51.110,160.121
C01274=1016.672,353.000,-150.545,171.150,51.114,160.120
C01275=1016.665,352.729,-150.505,171.141,51.118,160.120
C01276=1016.656,352.458,-150.463,171.132,51.121,160.119
C01277=1016.647,352.187,-150.423,171.124,51.124,160.118
C01278=1016.640,351.940,-150.386,171.116,51.127,160.118
C01279=1016.632,351.693,-150.349,171.108,51.130,160.117
C01280=1016.625,351.446,-150.312,171.100,51.132,160.116
C01281=1016.618,351.198,-150.275,171.092,51.135,160.115
C01282=1016.610,350.951,-150.238,171.085,51.139,160.115
C01283=1016.603,350.705,-150.201,171.077,51.142,160.114
C01284=1016.596,350.457,-150.164,171.069,51.145,160.113
C01285=1016.589,350.210,-150.127,171.061,51.148,160.113
C01286=1016.581,349.963,-150.091,171.053,51.151,160.112
C01287=1016.574,349.715,-150.053,171.045,51.154,160.112
C01288=1016.566,349.468,-150.017,171.037,51.157,160.111
C01289=1016.560,349.222,-149.980,171.029,51.160,160.110
C01290=1016.552,348.974,-149.944,171.022,51.163,160.110
C01291=1016.545,348.727,-149.906,171.013,51.166,160.109
C01292=1016.537,348.480,-149.870,171.006,51.170,160.108
C01293=1016.530,348.232,-149.832,170.998,51.173,160.108
C01294=1016.523,347.985,-149.796,170.990,51.176,160.107
C01295=1016.516,347.738,-149.760,170.982,51.179,160.106
C01296=1016.509,347.490,-149.723,170.975,51.182,160.106
C01297=1016.501,347.244,-149.686,170.968,51.185,160.105
C01298=1016.494,346.997,-149.650,170.960,51.188,160.104
C01299=1016.487,346.749,-149.613,170.952,51.192,160.104
C01300=1016.480,346.502,-149.577,170.945,51.195,160.103
C01301=1016.473,346.254,-149.541,170.937,51.198,160.103
C01302=1016.465,346.008,-149.504,170.929,51.202,160.102
C01303=1016.458,345.761,-149.468,170.921,51.205,160.102
C01304=1016.450,345.513,-149.432,170.913,51.208,160.101
C01305=1016.443,345.266,-149.395,170.906,51.212,160.100
C01306=1016.436,345.019,-149.359,170.898,51.215,160.100
C01307=1016.429,344.771,-149.323,170.891,51.218,160.099
C01308=1016.422,344.524,-149.287,170.884,51.222,160.099
C01309=1016.415,344.276,-149.251,170.876,51.225,160.098
C01310=1016.407,344.029,-149.215,170.868,51.229,160.098
C01311=1016.401,343.782,-149.178,170.861,51.232,160.097
C01312=1016.393,343.534,-149.142,170.853,51.235,160.096
C01313=1016.386,343.288,-149.106,170.845,51.239,160.096
C01314=1016.378,343.040,-149.070,170.839,51.242,160.096
C01315=1016.372,342.792,-149.034,170.831,51.245,160.095
C01316=1016.364,342.545,-148.998,170.823,51.249,160.095
C01317=1016.357,342.298,-148.962,170.816,51.253,160.094
C01318=1016.351,342.051,-148.927,170.808,51.256,160.093
C01319=1016.344,341.803,-148.890,170.801,51.260,160.093
C01320=1016.337,341.556,-148.854,170.793,51.263,160.092
C01321=1016.329,341.308,-148.819,170.786,51.266,160.092
C01322=1016.322,341.062,-148.783,170.779,51.270,160.092
C01323=1016.315,340.814,-148.748,170.771,51.274,160.091
C01324=1016.308,340.566,-148.711,170.764,51.277,160.090
C01325=1016.301,340.320,-148.675,170.756,51.281,160.090
C01326=1016.294,340.072,-148.640,170.748,51.284,160.089
C01327=1016.287,339.825,-148.604,170.742,51.288,160.089
C01328=1016.280,339.578,-148.569,170.735,51.292,160.089
C01329=1016.274,339.329,-148.532,170.727,51.295,160.088
C01330=1016.266,339.082,-148.497,170.719,51.299,160.088
C01331=1016.260,338.835,-148.461,170.712,51.302,160.087
C01332=1016.253,338.588,-148.426,170.706,51.306,160.087
C01333=1016.245,338.340,-148.390,170.698,51.310,160.086
C01334=1016.238,338.067,-148.352,170.689,51.314,160.086
C01335=1016.230,337.793,-148.312,170.681,51.318,160.085
C01336=1016.222,337.519,-148.273,170.674,51.322,160.085
C01337=1016.215,337.245,-148.234,170.665,51.326,160.084
C01338=1016.208,336.998,-148.199,170.658,51.330,160.084
C01339=1016.200,336.751,-148.164,170.651,51.334,160.084
C01340=1016.193,336.504,-148.128,170.644,51.337,160.083
C01341=1016.186,336.257,-148.093,170.637,51.341,160.083
C01342=1016.179,336.009,-148.058,170.629,51.345,160.082
C01343=1016.172,335.761,-148.023,170.622,51.349,160.082
C01344=1016.166,335.514,-147.988,170.615,51.352,160.082
C01345=1016.159,335.267,-147.952,170.608,51.357,160.081
C01346=1016.152,335.019,-147.917,170.601,51.360,160.081
C01347=1016.145,334.772,-147.882,170.594,51.364,160.080
C01348=1016.139,334.524,-147.848,170.586,51.369,160.080
C01349=1016.132,334.276,-147.813,170.580,51.372,160.080
C01350=1016.125,334.029,-147.777,170.573,51.376,160.079
C01351=1016.119,333.782,-147.742,170.565,51.380,160.079
C01352=1016.112,333.534,-147.707,170.558,51.384,160.079
C01353=1016.105,333.287,-147.672,170.552,51.388,160.078
C01354=1016.098,333.040,-147.637,170.544,51.392,160.078
C01355=1016.091,332.792,-147.603,170.537,51.395,160.078
C01356=1016.084,332.545,-147.568,170.530,51.400,160.077
C01357=1016.077,332.297,-147.533,170.523,51.404,160.077
C01358=1016.071,332.049,-147.498,170.516,51.408,160.077
C01359=1016.064,331.802,-147.463,170.509,51.412,160.076
C01360=1016.057,331.555,-147.429,170.501,51.416,160.076
C01361=1016.050,331.307,-147.394,170.494,51.420,160.076
C01362=1016.044,331.059,-147.359,170.488,51.424,160.075
C01363=1016.036,330.812,-147.325,170.481,51.428,160.075
C01364=1016.030,330.564,-147.290,170.474,51.432,160.075
C01365=1016.023,330.316,-147.256,170.466,51.436,160.074
C01366=1016.016,330.069,-147.221,170.460,51.440,160.074
C01367=1016.009,329.821,-147.187,170.453,51.444,160.074
C01368=1016.003,329.574,-147.153,170.446,51.449,160.074
C01369=1015.996,329.327,-147.118,170.439,51.453,160.073
C01370=1015.989,329.079,-147.084,170.433,51.457,160.073
C01371=1015.983,328.832,-147.049,170.425,51.461,160.073
C01372=1015.976,328.584,-147.014,170.418,51.465,160.072
C01373=1015.969,328.337,-146.981,170.411,51.469,160.072
C01374=1015.963,328.089,-146.946,170.405,51.474,160.072
C01375=1015.956,327.841,-146.911,170.398,51.478,160.072
C01376=1015.949,327.594,-146.877,170.391,51.482,160.071
C01377=1015.943,327.346,-146.843,170.384,51.486,160.071
C01378=1015.937,327.098,-146.809,170.377,51.490,160.071
C01379=1015.929,326.851,-146.774,170.370,51.495,160.071
C01380=1015.923,326.603,-146.740,170.364,51.499,160.070
C01381=1015.917,326.356,-146.706,170.356,51.504,160.070
C01382=1015.910,326.108,-146.672,170.350,51.507,160.070
C01383=1015.903,325.860,-146.638,170.343,51.512,160.070
C01384=1015.897,325.614,-146.604,170.336,51.517,160.070
C01385=1015.889,325.366,-146.570,170.329,51.521,160.069
C01386=1015.882,325.118,-146.537,170.323,51.525,160.069
C01387=1015.876,324.871,-146.503,170.316,51.530,160.069
C01388=1015.869,324.623,-146.469,170.309,51.534,160.069
C01389=1015.862,324.375,-146.436,170.302,51.539,160.068
C01390=1015.856,324.128,-146.402,170.295,51.544,160.068
C01391=1015.848,323.880,-146.368,170.289,51.547,160.068
C01392=1015.842,323.632,-146.334,170.282,51.552,160.068
C01393=1015.836,323.385,-146.301,170.276,51.557,160.068
C01394=1015.829,323.107,-146.263,170.267,51.562,160.067
C01395=1015.821,322.829,-146.226,170.261,51.567,160.067
C01396=1015.813,322.551,-146.188,170.253,51.572,160.067
C01397=1015.805,322.273,-146.150,170.245,51.577,160.067
C01398=1015.799,322.025,-146.117,170.238,51.582,160.067
C01399=1015.792,321.778,-146.083,170.233,51.587,160.067
C01400=1015.786,321.531,-146.050,170.225,51.591,160.067
C01401=1015.779,321.282,-146.016,170.219,51.596,160.066
C01402=1015.772,321.035,-145.983,170.212,51.601,160.066
C01403=1015.766,320.787,-145.949,170.206,51.605,160.066
C01404=1015.759,320.540,-145.916,170.199,51.609,160.066
C01405=1015.753,320.292,-145.883,170.192,51.614,160.066
C01406=1015.746,320.044,-145.849,170.185,51.619,160.066
C01407=1015.740,319.797,-145.816,170.180,51.624,160.066
C01408=1015.733,319.549,-145.782,170.173,51.629,160.066
C01409=1015.727,319.301,-145.749,170.166,51.633,160.065
C01410=1015.720,319.054,-145.716,170.159,51.638,160.065
C01411=1015.713,318.806,-145.683,170.153,51.642,160.065
C01412=1015.708,318.558,-145.649,170.146,51.647,160.065
C01413=1015.700,318.310,-145.616,170.140,51.652,160.065
C01414=1015.694,318.063,-145.583,170.133,51.657,160.065
C01415=1015.688,317.815,-145.550,170.127,51.661,160.065
C01416=1015.681,317.568,-145.517,170.120,51.666,160.065
C01417=1015.675,317.320,-145.483,170.114,51.671,160.065
C01418=1015.669,317.072,-145.450,170.108,51.676,160.065
C01419=1015.663,316.824,-145.417,170.101,51.681,160.065
C01420=1015.655,316.577,-145.384,170.094,51.686,160.064
C01421=1015.649,316.329,-145.351,170.087,51.691,160.064
C01422=1015.644,316.081,-145.318,170.082,51.695,160.064
C01423=1015.637,315.834,-145.285,170.075,51.700,160.064
C01424=1015.631,315.586,-145.252,170.068,51.705,160.064
C01425=1015.624,315.338,-145.218,170.062,51.709,160.064
C01426=1015.617,315.091,-145.186,170.056,51.714,160.064
C01427=1015.612,314.843,-145.152,170.049,51.719,160.064
C01428=1015.606,314.595,-145.119,170.042,51.724,160.064
C01429=1015.599,314.348,-145.087,170.037,51.729,160.064
C01430=1015.593,314.100,-145.054,170.030,51.734,160.064
C01431=1015.586,313.852,-145.021,170.023,51.739,160.064
C01432=1015.581,313.604,-144.988,170.017,51.744,160.064
C01433=1015.574,313.356,-144.955,170.011,51.749,160.063
C01434=1015.568,313.109,-144.922,170.004,51.754,160.064
C01435=1015.562,312.861,-144.889,169.999,51.759,160.064
C01436=1015.555,312.614,-144.857,169.992,51.764,160.063
C01437=1015.550,312.366,-144.823,169.985,51.769,160.063
C01438=1015.544,312.118,-144.790,169.980,51.774,160.064
C01439=1015.537,311.871,-144.758,169.973,51.779,160.063
C01440=1015.531,311.623,-144.725,169.966,51.784,160.063
C01441=1015.525,311.375,-144.692,169.961,51.789,160.064
C01442=1015.519,311.127,-144.660,169.954,51.794,160.063
C01443=1015.513,310.879,-144.627,169.947,51.799,160.063
C01444=1015.507,310.632,-144.594,169.942,51.804,160.063
C01445=1015.501,310.384,-144.561,169.935,51.809,160.063
C01446=1015.494,310.136,-144.529,169.929,51.814,160.063
C01447=1015.488,309.888,-144.497,169.923,51.819,160.063
C01448=1015.483,309.640,-144.463,169.917,51.824,160.064
C01449=1015.476,309.393,-144.431,169.910,51.829,160.063
C01450=1015.470,309.146,-144.399,169.904,51.835,160.063
C01451=1015.464,308.898,-144.367,169.898,51.840,160.063
C01452=1015.457,308.650,-144.335,169.892,51.845,160.064
C01453=1015.451,308.402,-144.303,169.885,51.851,160.064
C01454=1015.444,308.130,-144.268,169.878,51.857,160.064
C01455=1015.436,307.858,-144.232,169.872,51.862,160.064
C01456=1015.430,307.585,-144.197,169.864,51.868,160.064
C01457=1015.423,307.312,-144.162,169.858,51.874,160.064
C01458=1015.417,307.064,-144.130,169.852,51.879,160.064
C01459=1015.410,306.817,-144.098,169.845,51.885,160.064
C01460=1015.404,306.569,-144.066,169.839,51.891,160.064
C01461=1015.397,306.321,-144.035,169.834,51.896,160.064
C01462=1015.391,306.073,-144.003,169.827,51.901,160.064
C01463=1015.385,305.825,-143.971,169.821,51.907,160.065
C01464=1015.379,305.578,-143.939,169.814,51.912,160.064
C01465=1015.372,305.330,-143.907,169.808,51.918,160.064
C01466=1015.366,305.082,-143.875,169.803,51.923,160.065
C01467=1015.359,304.834,-143.844,169.796,51.928,160.065
C01468=1015.353,304.586,-143.812,169.790,51.934,160.065
C01469=1015.347,304.338,-143.781,169.784,51.940,160.065
C01470=1015.341,304.090,-143.749,169.777,51.945,160.065
C01471=1015.335,303.842,-143.717,169.772,51.950,160.065
C01472=1015.329,303.594,-143.685,169.766,51.956,160.065
C01473=1015.323,303.347,-143.653,169.759,51.962,160.065
C01474=1015.316,303.099,-143.621,169.753,51.967,160.066
C01475=1015.311,302.850,-143.590,169.748,51.972,160.066
C01476=1015.304,302.603,-143.559,169.742,51.979,160.066
C01477=1015.298,302.355,-143.527,169.735,51.984,160.066
C01478=1015.292,302.107,-143.496,169.729,51.990,160.066
C01479=1015.286,301.859,-143.464,169.723,51.996,160.066
C01480=1015.280,301.612,-143.433,169.717,52.001,160.066
C01481=1015.274,301.363,-143.401,169.711,52.006,160.067
C01482=1015.267,301.116,-143.369,169.705,52.012,160.067
C01483=1015.262,300.868,-143.337,169.699,52.018,160.067
C01484=1015.256,300.620,-143.305,169.693,52.024,160.067
C01485=1015.249,300.373,-143.274,169.687,52.029,160.067
C01486=1015.244,300.124,-143.243,169.681,52.035,160.067
C01487=1015.237,299.876,-143.212,169.674,52.040,160.067
C01488=1015.232,299.628,-143.180,169.670,52.046,160.068
C01489=1015.225,299.380,-143.149,169.663,52.052,160.068
C01490=1015.220,299.132,-143.118,169.657,52.058,160.068
C01491=1015.213,298.884,-143.086,169.651,52.064,160.068
C01492=1015.208,298.637,-143.054,169.645,52.069,160.068
C01493=1015.201,298.389,-143.023,169.639,52.075,160.069
C01494=1015.196,298.141,-142.992,169.633,52.081,160.069
C01495=1015.189,297.893,-142.961,169.627,52.087,160.069
C01496=1015.184,297.646,-142.929,169.621,52.092,160.069
C01497=1015.177,297.397,-142.898,169.616,52.098,160.069
C01498=1015.172,297.149,-142.867,169.610,52.104,160.070
C01499=1015.166,296.901,-142.836,169.604,52.110,160.070
C01500=1015.160,296.653,-142.804,169.597,52.116,160.070
C01501=1015.154,296.405,-142.772,169.592,52.121,160.070
C01502=1015.148,296.157,-142.742,169.586,52.127,160.070
C01503=1015.142,295.909,-142.710,169.580,52.133,160.071
C01504=1015.137,295.661,-142.679,169.574,52.139,160.071
C01505=1015.131,295.414,-142.648,169.568,52.145,160.071
C01506=1015.125,295.165,-142.617,169.563,52.151,160.071
C01507=1015.119,294.918,-142.585,169.556,52.156,160.071
C01508=1015.113,294.669,-142.555,169.551,52.163,160.072
C01509=1015.108,294.422,-142.523,169.545,52.169,160.072
C01510=1015.102,294.174,-142.493,169.539,52.174,160.072
C01511=1015.096,293.926,-142.461,169.534,52.181,160.072
C01512=1015.090,293.678,-142.430,169.527,52.186,160.073
C01513=1015.085,293.430,-142.399,169.521,52.192,160.073
C01514=1015.079,293.175,-142.367,169.515,52.199,160.073
C01515=1015.073,292.921,-142.335,169.509,52.204,160.073
C01516=1015.067,292.666,-142.304,169.504,52.210,160.074
C01517=1015.060,292.412,-142.272,169.497,52.217,160.074
C01518=1015.054,292.164,-142.242,169.492,52.223,160.074
C01519=1015.049,291.916,-142.211,169.487,52.229,160.075
C01520=1015.043,291.667,-142.180,169.481,52.236,160.075
C01521=1015.037,291.420,-142.150,169.475,52.242,160.075
C01522=1015.031,291.172,-142.119,169.468,52.248,160.075
C01523=1015.025,290.924,-142.089,169.463,52.254,160.076
C01524=1015.020,290.675,-142.058,169.458,52.260,160.076
C01525=1015.014,290.427,-142.027,169.452,52.266,160.076
C01526=1015.008,290.179,-141.997,169.446,52.272,160.077
C01527=1015.002,289.932,-141.967,169.440,52.279,160.077
C01528=1014.996,289.683,-141.936,169.434,52.285,160.077
C01529=1014.990,289.435,-141.905,169.428,52.291,160.077
C01530=1014.984,289.187,-141.875,169.422,52.298,160.078
C01531=1014.978,288.940,-141.845,169.417,52.304,160.078
C01532=1014.972,288.691,-141.814,169.412,52.310,160.078
C01533=1014.966,288.443,-141.784,169.406,52.316,160.079
C01534=1014.961,288.195,-141.754,169.400,52.323,160.079
C01535=1014.955,287.947,-141.724,169.394,52.329,160.079
C01536=1014.949,287.699,-141.693,169.389,52.336,160.080
C01537=1014.943,287.451,-141.663,169.383,52.342,160.080
C01538=1014.937,287.203,-141.632,169.377,52.349,160.080
C01539=1014.931,286.954,-141.603,169.371,52.355,160.081
C01540=1014.926,286.707,-141.572,169.366,52.361,160.081
C01541=1014.920,286.459,-141.542,169.360,52.367,160.081
C01542=1014.914,286.211,-141.512,169.355,52.374,160.082
C01543=1014.908,285.962,-141.482,169.349,52.381,160.082
C01544=1014.903,285.715,-141.452,169.343,52.387,160.083
C01545=1014.897,285.466,-141.422,169.337,52.393,160.083
C01546=1014.891,285.218,-141.392,169.332,52.400,160.083
C01547=1014.885,284.971,-141.361,169.326,52.407,160.084
C01548=1014.880,284.722,-141.332,169.320,52.413,160.084
C01549=1014.873,284.474,-141.301,169.315,52.420,160.084
C01550=1014.867,284.225,-141.272,169.310,52.426,160.085
C01551=1014.861,283.978,-141.242,169.304,52.432,160.085
C01552=1014.856,283.729,-141.212,169.299,52.439,160.086
C01553=1014.850,283.481,-141.182,169.293,52.446,160.086
C01554=1014.844,283.233,-141.153,169.287,52.453,160.086
C01555=1014.838,282.985,-141.122,169.281,52.459,160.087
C01556=1014.833,282.737,-141.093,169.276,52.466,160.087
C01557=1014.827,282.489,-141.063,169.270,52.473,160.088
C01558=1014.820,282.241,-141.033,169.265,52.480,160.088
C01559=1014.815,281.993,-141.004,169.259,52.486,160.088
C01560=1014.809,281.744,-140.974,169.253,52.493,160.089
C01561=1014.803,281.497,-140.944,169.248,52.499,160.089
C01562=1014.798,281.249,-140.915,169.242,52.506,160.090
C01563=1014.792,281.000,-140.885,169.237,52.513,160.090
C01564=1014.787,280.752,-140.856,169.231,52.520,160.090
C01565=1014.780,280.505,-140.826,169.225,52.527,160.091
C01566=1014.775,280.256,-140.796,169.220,52.533,160.091
C01567=1014.769,280.008,-140.767,169.214,52.540,160.092
C01568=1014.763,279.760,-140.738,169.209,52.547,160.092
C01569=1014.758,279.511,-140.708,169.203,52.554,160.093
C01570=1014.753,279.266,-140.678,169.198,52.561,160.093
C01571=1014.746,279.021,-140.649,169.192,52.568,160.094
C01572=1014.740,278.776,-140.620,169.187,52.574,160.094
C01573=1014.736,278.530,-140.591,169.182,52.581,160.095
C01574=1014.729,278.285,-140.562,169.176,52.588,160.095
C01575=1014.724,278.040,-140.532,169.171,52.594,160.095
C01576=1014.718,277.795,-140.503,169.165,52.601,160.096
C01577=1014.713,277.550,-140.475,169.160,52.608,160.096
C01578=1014.708,277.302,-140.445,169.154,52.615,160.097
C01579=1014.701,277.053,-140.416,169.149,52.622,160.097
C01580=1014.696,276.806,-140.387,169.143,52.629,160.098
C01581=1014.691,276.557,-140.357,169.138,52.636,160.098
C01582=1014.685,276.309,-140.327,169.132,52.643,160.099
C01583=1014.679,276.061,-140.298,169.127,52.650,160.099
C01584=1014.674,275.813,-140.269,169.122,52.657,160.100
C01585=1014.668,275.565,-140.240,169.116,52.664,160.100
C01586=1014.662,275.316,-140.210,169.111,52.671,160.101
C01587=1014.656,275.068,-140.181,169.105,52.678,160.101
C01588=1014.651,274.820,-140.152,169.100,52.685,160.102
C01589=1014.645,274.572,-140.124,169.095,52.692,160.102
C01590=1014.640,274.323,-140.094,169.089,52.699,160.103
C01591=1014.634,274.075,-140.065,169.084,52.706,160.103
C01592=1014.628,273.828,-140.036,169.078,52.713,160.104
C01593=1014.623,273.579,-140.008,169.073,52.721,160.104
C01594=1014.616,273.331,-139.979,169.068,52.728,160.105
C01595=1014.612,273.083,-139.949,169.062,52.735,160.105
C01596=1014.606,272.834,-139.921,169.057,52.742,160.106
C01597=1014.600,272.586,-139.891,169.050,52.749,160.106
C01598=1014.594,272.338,-139.863,169.045,52.756,160.107
C01599=1014.589,272.089,-139.834,169.040,52.764,160.107
C01600=1014.583,271.841,-139.805,169.035,52.771,160.108
C01601=1014.578,271.593,-139.777,169.029,52.778,160.108
C01602=1014.572,271.344,-139.747,169.024,52.785,160.109
C01603=1014.566,271.096,-139.718,169.019,52.792,160.109
C01604=1014.561,270.848,-139.689,169.014,52.800,160.110
C01605=1014.555,270.600,-139.660,169.008,52.807,160.111
C01606=1014.550,270.352,-139.632,169.003,52.814,160.111
C01607=1014.544,270.103,-139.603,168.998,52.822,160.112
C01608=1014.539,269.855,-139.575,168.992,52.830,160.112
C01609=1014.533,269.607,-139.546,168.986,52.837,160.113
C01610=1014.527,269.358,-139.517,168.981,52.844,160.114
C01611=1014.522,269.110,-139.489,168.976,52.852,160.114
C01612=1014.516,268.862,-139.460,168.970,52.859,160.115
C01613=1014.511,268.614,-139.431,168.966,52.866,160.115
C01614=1014.505,268.365,-139.402,168.960,52.874,160.116
C01615=1014.500,268.117,-139.374,168.955,52.881,160.117
C01616=1014.494,267.869,-139.346,168.949,52.889,160.117
C01617=1014.489,267.620,-139.317,168.944,52.897,160.118
C01618=1014.483,267.372,-139.288,168.939,52.904,160.118
C01619=1014.477,267.124,-139.260,168.934,52.911,160.119
C01620=1014.472,266.875,-139.232,168.928,52.919,160.119
C01621=1014.466,266.627,-139.204,168.923,52.926,160.120
C01622=1014.461,266.379,-139.175,168.917,52.934,160.121
C01623=1014.455,266.131,-139.147,168.912,52.942,160.121
C01624=1014.449,265.882,-139.118,168.907,52.949,160.122
C01625=1014.444,265.634,-139.090,168.902,52.957,160.123
C01626=1014.438,265.385,-139.062,168.897,52.964,160.123
C01627=1014.434,265.137,-139.033,168.892,52.971,160.124
C01628=1014.428,264.889,-139.005,168.886,52.980,160.124
C01629=1014.422,264.641,-138.976,168.880,52.987,160.125
C01630=1014.417,264.397,-138.950,168.875,52.995,160.126
C01631=1014.412,264.155,-138.922,168.870,53.002,160.126
C01632=1014.406,263.911,-138.894,168.865,53.009,160.127
C01633=1014.400,263.669,-138.867,168.860,53.017,160.128
C01634=1014.395,263.426,-138.840,168.855,53.024,160.128
C01635=1014.390,263.183,-138.812,168.850,53.032,160.129
C01636=1014.384,262.941,-138.785,168.845,53.040,160.130
C01637=1014.378,262.697,-138.757,168.840,53.047,160.130
C01638=1014.373,262.449,-138.729,168.834,53.055,160.131
C01639=1014.368,262.201,-138.701,168.829,53.063,160.131
C01640=1014.362,261.952,-138.673,168.824,53.071,160.132
C01641=1014.357,261.704,-138.645,168.819,53.079,160.133
C01642=1014.351,261.456,-138.617,168.813,53.087,160.133
C01643=1014.345,261.207,-138.589,168.808,53.094,160.134
C01644=1014.340,260.959,-138.561,168.803,53.102,160.135
C01645=1014.335,260.711,-138.533,168.798,53.110,160.135
C01646=1014.329,260.462,-138.505,168.792,53.118,160.136
C01647=1014.324,260.213,-138.478,168.787,53.126,160.137
C01648=1014.318,259.965,-138.450,168.782,53.134,160.137
C01649=1014.313,259.717,-138.422,168.778,53.141,160.138
C01650=1014.308,259.468,-138.393,168.772,53.150,160.139
C01651=1014.302,259.220,-138.366,168.767,53.157,160.140
C01652=1014.297,258.972,-138.338,168.762,53.165,160.140
C01653=1014.291,258.724,-138.311,168.756,53.174,160.141
C01654=1014.286,258.475,-138.284,168.752,53.182,160.142
C01655=1014.279,258.227,-138.256,168.747,53.190,160.143
C01656=1014.274,257.978,-138.229,168.741,53.198,160.143
C01657=1014.268,257.730,-138.201,168.736,53.206,160.144
C01658=1014.263,257.482,-138.174,168.730,53.214,160.145
C01659=1014.257,257.232,-138.146,168.726,53.223,160.146
C01660=1014.251,256.985,-138.119,168.721,53.231,160.146
C01661=1014.246,256.736,-138.092,168.715,53.239,160.147
C01662=1014.241,256.488,-138.064,168.710,53.247,160.148
C01663=1014.235,256.240,-138.037,168.705,53.256,160.148
C01664=1014.229,255.990,-138.010,168.700,53.263,160.149
C01665=1014.224,255.742,-137.982,168.694,53.272,160.150
C01666=1014.218,255.494,-137.955,168.689,53.280,160.151
C01667=1014.213,255.246,-137.927,168.685,53.288,160.151
C01668=1014.207,254.997,-137.900,168.679,53.296,160.152
C01669=1014.202,254.749,-137.873,168.674,53.305,160.153
C01670=1014.196,254.499,-137.845,168.668,53.313,160.154
C01671=1014.190,254.252,-137.818,168.664,53.321,160.154
C01672=1014.185,254.003,-137.791,168.658,53.330,160.155
C01673=1014.179,253.755,-137.764,168.653,53.338,160.156
C01674=1014.174,253.507,-137.736,168.649,53.346,160.157
C01675=1014.168,253.258,-137.710,168.643,53.354,160.158
C01676=1014.163,253.010,-137.682,168.639,53.363,160.158
C01677=1014.158,252.761,-137.655,168.633,53.371,160.159
C01678=1014.152,252.513,-137.628,168.628,53.380,160.160
C01679=1014.147,252.264,-137.601,168.623,53.388,160.161
C01680=1014.141,252.016,-137.574,168.618,53.396,160.161
C01681=1014.136,251.767,-137.547,168.612,53.405,160.162
C01682=1014.131,251.518,-137.519,168.608,53.413,160.163
C01683=1014.125,251.270,-137.492,168.602,53.422,160.164
C01684=1014.120,251.021,-137.465,168.598,53.430,160.165
C01685=1014.114,250.773,-137.438,168.593,53.438,160.165
C01686=1014.109,250.525,-137.411,168.587,53.447,160.166
C01687=1014.104,250.276,-137.383,168.583,53.455,160.167
C01688=1014.098,250.028,-137.357,168.577,53.464,160.168
C01689=1014.093,249.779,-137.329,168.573,53.473,160.169
C01690=1014.088,249.535,-137.303,168.567,53.481,160.169
C01691=1014.083,249.292,-137.277,168.562,53.489,160.170
C01692=1014.078,249.047,-137.250,168.558,53.497,160.171
C01693=1014.072,248.804,-137.224,168.552,53.506,160.172
C01694=1014.066,248.560,-137.197,168.548,53.514,160.173
C01695=1014.062,248.316,-137.171,168.543,53.523,160.174
C01696=1014.057,248.072,-137.145,168.537,53.531,160.174
C01697=1014.051,247.828,-137.118,168.533,53.540,160.175
C01698=1014.046,247.579,-137.091,168.527,53.548,160.176
C01699=1014.040,247.331,-137.064,168.523,53.557,160.177
C01700=1014.036,247.083,-137.037,168.517,53.565,160.178
C01701=1014.030,246.835,-137.010,168.513,53.574,160.179
C01702=1014.025,246.586,-136.983,168.507,53.582,160.179
C01703=1014.020,246.337,-136.956,168.503,53.591,160.180
C01704=1014.015,246.088,-136.930,168.498,53.600,160.181
C01705=1014.010,245.840,-136.903,168.493,53.609,160.182
C01706=1014.004,245.591,-136.876,168.487,53.617,160.183
C01707=1013.999,245.343,-136.849,168.483,53.625,160.184
C01708=1013.994,245.095,-136.822,168.478,53.634,160.184
C01709=1013.989,244.846,-136.795,168.473,53.643,160.185
C01710=1013.984,244.597,-136.769,168.468,53.652,160.186
C01711=1013.978,244.349,-136.742,168.464,53.661,160.187
C01712=1013.974,244.101,-136.715,168.458,53.670,160.188
C01713=1013.968,243.852,-136.689,168.454,53.678,160.189
C01714=1013.963,243.604,-136.661,168.448,53.687,160.190
C01715=1013.958,243.354,-136.635,168.444,53.695,160.190
C01716=1013.952,243.106,-136.608,168.439,53.704,160.191
C01717=1013.948,242.858,-136.581,168.433,53.713,160.192
C01718=1013.942,242.610,-136.555,168.429,53.722,160.193
C01719=1013.937,242.360,-136.528,168.423,53.731,160.194
C01720=1013.932,242.113,-136.502,168.419,53.739,160.195
C01721=1013.927,241.864,-136.476,168.414,53.749,160.196
C01722=1013.921,241.615,-136.449,168.409,53.758,160.197
C01723=1013.917,241.367,-136.423,168.405,53.767,160.198
C01724=1013.911,241.119,-136.397,168.399,53.776,160.199
C01725=1013.906,240.870,-136.371,168.394,53.785,160.199
C01726=1013.901,240.621,-136.343,168.390,53.794,160.200
C01727=1013.896,240.373,-136.318,168.384,53.803,160.201
C01728=1013.890,240.124,-136.291,168.379,53.812,160.202
C01729=1013.885,239.875,-136.265,168.375,53.820,160.203
C01730=1013.880,239.627,-136.238,168.370,53.830,160.204
C01731=1013.875,239.378,-136.212,168.365,53.839,160.205
C01732=1013.869,239.130,-136.186,168.360,53.848,160.206
C01733=1013.865,238.881,-136.160,168.355,53.857,160.207
C01734=1013.859,238.632,-136.134,168.350,53.866,160.208
C01735=1013.853,238.384,-136.107,168.345,53.875,160.209
C01736=1013.849,238.136,-136.081,168.341,53.884,160.210
C01737=1013.843,237.887,-136.056,168.336,53.894,160.211
C01738=1013.838,237.639,-136.029,168.330,53.903,160.212
C01739=1013.832,237.390,-136.003,168.325,53.912,160.212
C01740=1013.827,237.141,-135.977,168.321,53.921,160.214
C01741=1013.822,236.893,-135.952,168.316,53.930,160.214
C01742=1013.817,236.644,-135.926,168.311,53.940,160.216
C01743=1013.811,236.395,-135.900,168.306,53.949,160.216
C01744=1013.806,236.147,-135.874,168.301,53.959,160.217
C01745=1013.801,235.898,-135.848,168.297,53.968,160.218
C01746=1013.796,235.650,-135.822,168.292,53.977,160.220
C01747=1013.790,235.401,-135.796,168.287,53.986,160.220
C01748=1013.785,235.153,-135.771,168.282,53.996,160.221
C01749=1013.780,234.904,-135.745,168.277,54.005,160.222
C01750=1013.775,234.657,-135.719,168.272,54.015,160.223
C01751=1013.769,234.409,-135.693,168.267,54.024,160.224
C01752=1013.764,234.162,-135.668,168.263,54.033,160.225
C01753=1013.759,233.915,-135.642,168.257,54.042,160.226
C01754=1013.753,233.667,-135.617,168.253,54.052,160.227
C01755=1013.749,233.420,-135.591,168.247,54.061,160.228
C01756=1013.743,233.172,-135.566,168.243,54.071,160.229
C01757=1013.739,232.925,-135.540,168.239,54.080,160.230
C01758=1013.733,232.676,-135.514,168.233,54.090,160.231
C01759=1013.728,232.428,-135.488,168.229,54.099,160.232
C01760=1013.723,232.179,-135.462,168.224,54.109,160.233
C01761=1013.718,231.930,-135.437,168.219,54.118,160.234
C01762=1013.713,231.681,-135.412,168.214,54.128,160.235
C01763=1013.707,231.433,-135.387,168.210,54.137,160.237
C01764=1013.702,231.185,-135.361,168.205,54.146,160.237
C01765=1013.697,230.936,-135.335,168.200,54.156,160.238
C01766=1013.692,230.688,-135.309,168.195,54.166,160.240
C01767=1013.686,230.439,-135.284,168.190,54.176,160.241
C01768=1013.682,230.191,-135.258,168.185,54.185,160.241
C01769=1013.676,229.941,-135.233,168.180,54.195,160.243
C01770=1013.672,229.693,-135.207,168.176,54.205,160.244
C01771=1013.667,229.444,-135.182,168.171,54.214,160.245
C01772=1013.661,229.195,-135.156,168.166,54.223,160.246
C01773=1013.656,228.947,-135.131,168.161,54.233,160.247
C01774=1013.651,228.699,-135.106,168.156,54.243,160.248
C01775=1013.646,228.450,-135.080,168.151,54.253,160.249
C01776=1013.641,228.201,-135.055,168.147,54.263,160.250
C01777=1013.636,227.952,-135.029,168.142,54.272,160.251
